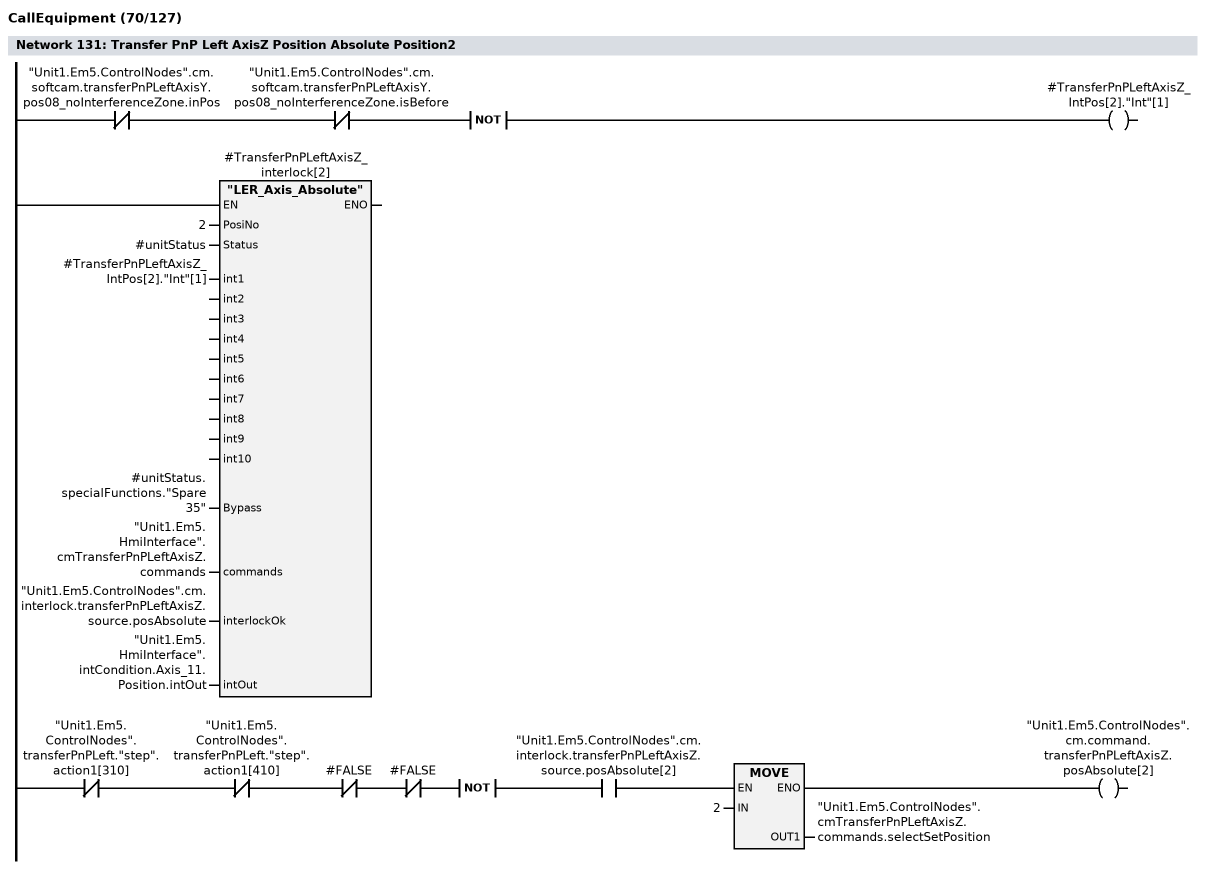
   RUNG wire#powerrail
      I_Contact( "Unit1.Em5.ControlNodes".cm.softcam.transferPnPLeftAxisY.pos08_noInterferenceZone.inPos )
      I_Contact( "Unit1.Em5.ControlNodes".cm.softcam.transferPnPLeftAxisY.pos08_noInterferenceZone.isBefore )
      Not()
      Coil( #TransferPnPLeftAxisZ_IntPos[2]."Int"[1] )
   END_RUNG
   RUNG wire#powerrail
      #TransferPnPLeftAxisZ_interlock[2](PosiNo := 2, Status := #unitStatus, int1 := #TransferPnPLeftAxisZ_IntPos[2]."Int"[1], int2 :=, int3 :=, int4 :=, int5 :=, int6 :=, int7 :=, int8 :=, int9 :=, int10 :=, Bypass := #unitStatus.specialFunctions."Spare 35", commands := "Unit1.Em5.HmiInterface".cmTransferPnPLeftAxisZ.commands, interlockOk := "Unit1.Em5.ControlNodes".cm.interlock.transferPnPLeftAxisZ.source.posAbsolute, intOut := "Unit1.Em5.HmiInterface".intCondition.Axis_11.Position.intOut)
   END_RUNG
   RUNG wire#powerrail
      I_Contact( "Unit1.Em5.ControlNodes".transferPnPLeft."step".action1[310] )
      I_Contact( "Unit1.Em5.ControlNodes".transferPnPLeft."step".action1[410] )
      I_Contact( #FALSE )
      I_Contact( #FALSE )
      Not()
      Contact( "Unit1.Em5.ControlNodes".cm.interlock.transferPnPLeftAxisZ.source.posAbsolute[2] )
      Move(in := 2, out1 => "Unit1.Em5.ControlNodes".cmTransferPnPLeftAxisZ.commands.selectSetPosition)
      Coil( "Unit1.Em5.ControlNodes".cm.command.transferPnPLeftAxisZ.posAbsolute[2] )
   END_RUNG
   // the same network as SCL:
   #TransferPnPLeftAxisZ_IntPos[2]."Int"[1] := NOT (NOT "Unit1.Em5.ControlNodes".cm.softcam.transferPnPLeftAxisY.pos08_noInterferenceZone.inPos AND NOT "Unit1.Em5.ControlNodes".cm.softcam.transferPnPLeftAxisY.pos08_noInterferenceZone.isBefore);
   #TransferPnPLeftAxisZ_interlock[2](PosiNo := 2,   // "LER_Axis_Absolute"
                           Status := #unitStatus,
                           int1 := #TransferPnPLeftAxisZ_IntPos[2]."Int"[1],
                           Bypass := #unitStatus.specialFunctions."Spare 35",
                           commands := "Unit1.Em5.HmiInterface".cmTransferPnPLeftAxisZ.commands,
                           interlockOk := "Unit1.Em5.ControlNodes".cm.interlock.transferPnPLeftAxisZ.source.posAbsolute,
                           intOut := "Unit1.Em5.HmiInterface".intCondition.Axis_11.Position.intOut);
   #_w1 := NOT (NOT "Unit1.Em5.ControlNodes".transferPnPLeft."step".action1[310] AND NOT "Unit1.Em5.ControlNodes".transferPnPLeft."step".action1[410] AND NOT #FALSE AND NOT #FALSE) AND "Unit1.Em5.ControlNodes".cm.interlock.transferPnPLeftAxisZ.source.posAbsolute[2];
   IF #_w1 THEN "Unit1.Em5.ControlNodes".cmTransferPnPLeftAxisZ.commands.selectSetPosition := 2; END_IF;
   "Unit1.Em5.ControlNodes".cm.command.transferPnPLeftAxisZ.posAbsolute[2] := #_w1;
END_REGION

REGION Network 132: Transfer PnP Left AxisZ Position Absolute Position3
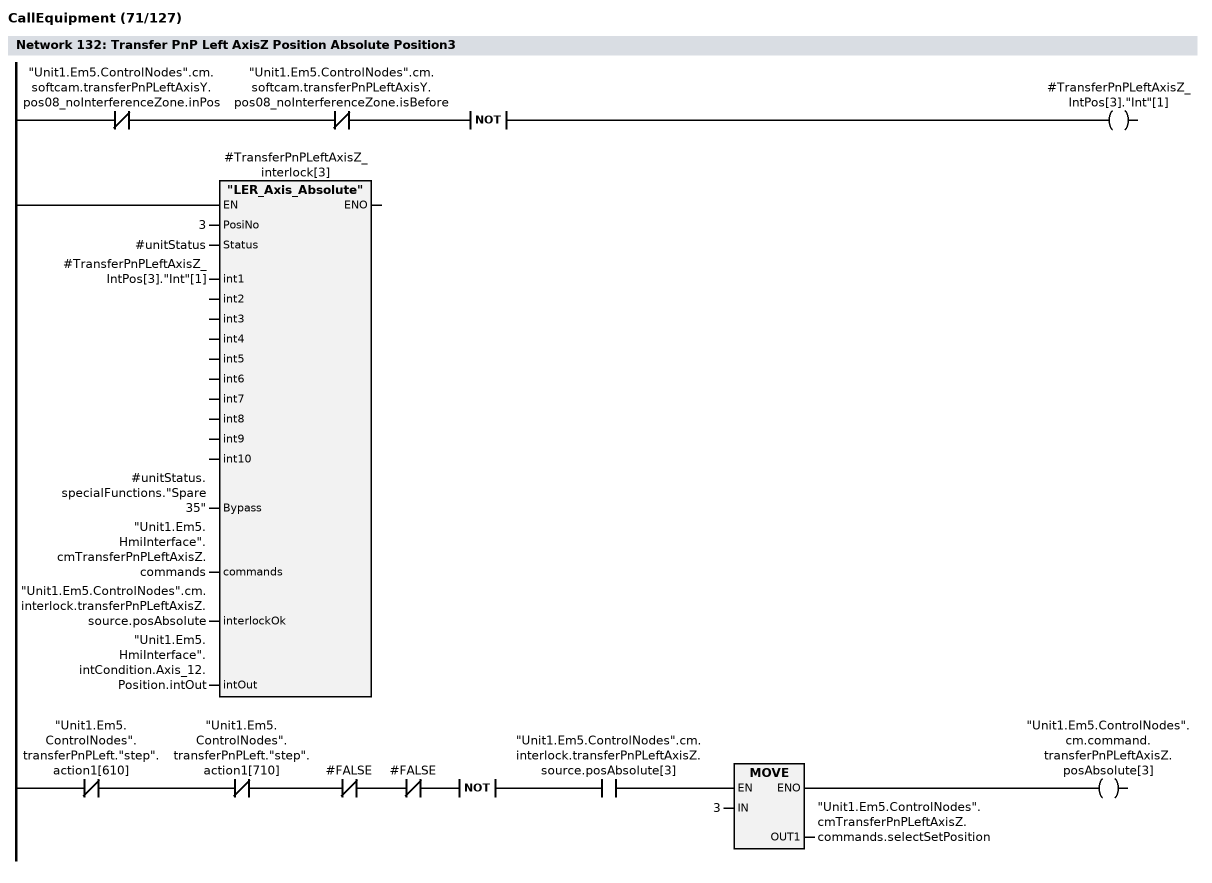
   RUNG wire#powerrail
      I_Contact( "Unit1.Em5.ControlNodes".cm.softcam.transferPnPLeftAxisY.pos08_noInterferenceZone.inPos )
      I_Contact( "Unit1.Em5.ControlNodes".cm.softcam.transferPnPLeftAxisY.pos08_noInterferenceZone.isBefore )
      Not()
      Coil( #TransferPnPLeftAxisZ_IntPos[3]."Int"[1] )
   END_RUNG
   RUNG wire#powerrail
      #TransferPnPLeftAxisZ_interlock[3](PosiNo := 3, Status := #unitStatus, int1 := #TransferPnPLeftAxisZ_IntPos[3]."Int"[1], int2 :=, int3 :=, int4 :=, int5 :=, int6 :=, int7 :=, int8 :=, int9 :=, int10 :=, Bypass := #unitStatus.specialFunctions."Spare 35", commands := "Unit1.Em5.HmiInterface".cmTransferPnPLeftAxisZ.commands, interlockOk := "Unit1.Em5.ControlNodes".cm.interlock.transferPnPLeftAxisZ.source.posAbsolute, intOut := "Unit1.Em5.HmiInterface".intCondition.Axis_12.Position.intOut)
   END_RUNG
   RUNG wire#powerrail
      I_Contact( "Unit1.Em5.ControlNodes".transferPnPLeft."step".action1[610] )
      I_Contact( "Unit1.Em5.ControlNodes".transferPnPLeft."step".action1[710] )
      I_Contact( #FALSE )
      I_Contact( #FALSE )
      Not()
      Contact( "Unit1.Em5.ControlNodes".cm.interlock.transferPnPLeftAxisZ.source.posAbsolute[3] )
      Move(in := 3, out1 => "Unit1.Em5.ControlNodes".cmTransferPnPLeftAxisZ.commands.selectSetPosition)
      Coil( "Unit1.Em5.ControlNodes".cm.command.transferPnPLeftAxisZ.posAbsolute[3] )
   END_RUNG
   // the same network as SCL:
   #TransferPnPLeftAxisZ_IntPos[3]."Int"[1] := NOT (NOT "Unit1.Em5.ControlNodes".cm.softcam.transferPnPLeftAxisY.pos08_noInterferenceZone.inPos AND NOT "Unit1.Em5.ControlNodes".cm.softcam.transferPnPLeftAxisY.pos08_noInterferenceZone.isBefore);
   #TransferPnPLeftAxisZ_interlock[3](PosiNo := 3,   // "LER_Axis_Absolute"
                           Status := #unitStatus,
                           int1 := #TransferPnPLeftAxisZ_IntPos[3]."Int"[1],
                           Bypass := #unitStatus.specialFunctions."Spare 35",
                           commands := "Unit1.Em5.HmiInterface".cmTransferPnPLeftAxisZ.commands,
                           interlockOk := "Unit1.Em5.ControlNodes".cm.interlock.transferPnPLeftAxisZ.source.posAbsolute,
                           intOut := "Unit1.Em5.HmiInterface".intCondition.Axis_12.Position.intOut);
   #_w1 := NOT (NOT "Unit1.Em5.ControlNodes".transferPnPLeft."step".action1[610] AND NOT "Unit1.Em5.ControlNodes".transferPnPLeft."step".action1[710] AND NOT #FALSE AND NOT #FALSE) AND "Unit1.Em5.ControlNodes".cm.interlock.transferPnPLeftAxisZ.source.posAbsolute[3];
   IF #_w1 THEN "Unit1.Em5.ControlNodes".cmTransferPnPLeftAxisZ.commands.selectSetPosition := 3; END_IF;
   "Unit1.Em5.ControlNodes".cm.command.transferPnPLeftAxisZ.posAbsolute[3] := #_w1;
END_REGION

REGION Network 133: Transfer PnP Left AxisZ Position Absolute Position4
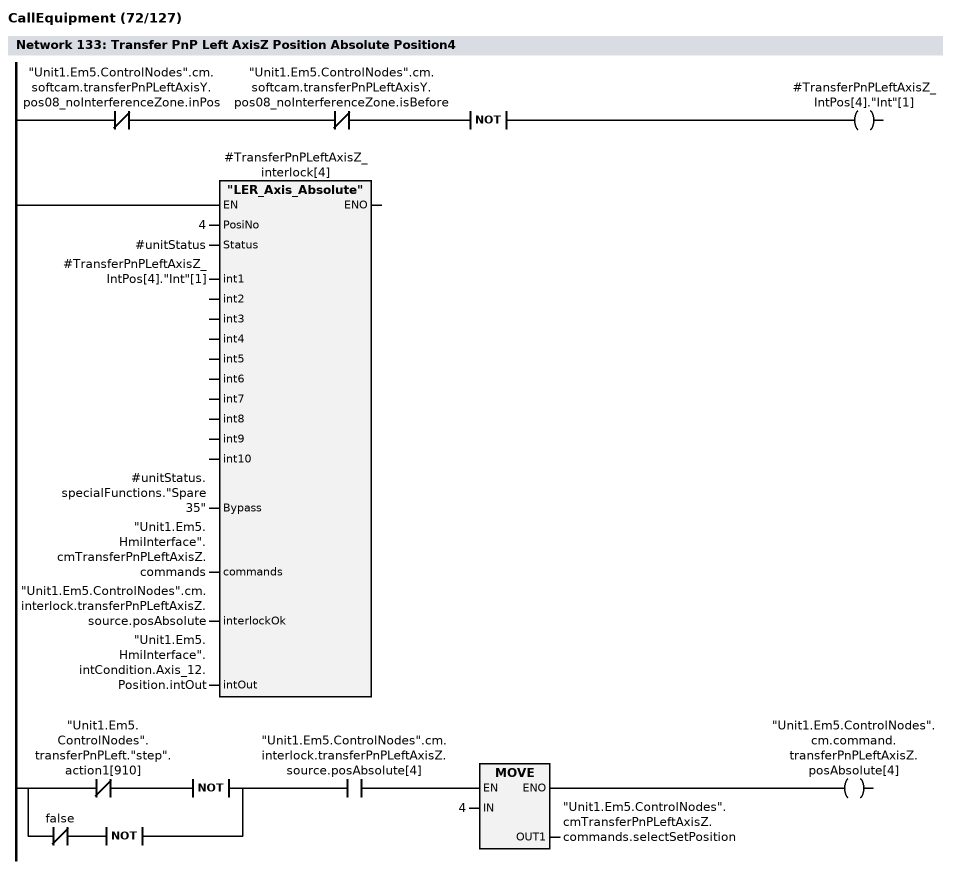
   RUNG wire#powerrail
      I_Contact( "Unit1.Em5.ControlNodes".cm.softcam.transferPnPLeftAxisY.pos08_noInterferenceZone.inPos )
      I_Contact( "Unit1.Em5.ControlNodes".cm.softcam.transferPnPLeftAxisY.pos08_noInterferenceZone.isBefore )
      Not()
      Coil( #TransferPnPLeftAxisZ_IntPos[4]."Int"[1] )
   END_RUNG
   RUNG wire#powerrail
      #TransferPnPLeftAxisZ_interlock[4](PosiNo := 4, Status := #unitStatus, int1 := #TransferPnPLeftAxisZ_IntPos[4]."Int"[1], int2 :=, int3 :=, int4 :=, int5 :=, int6 :=, int7 :=, int8 :=, int9 :=, int10 :=, Bypass := #unitStatus.specialFunctions."Spare 35", commands := "Unit1.Em5.HmiInterface".cmTransferPnPLeftAxisZ.commands, interlockOk := "Unit1.Em5.ControlNodes".cm.interlock.transferPnPLeftAxisZ.source.posAbsolute, intOut := "Unit1.Em5.HmiInterface".intCondition.Axis_12.Position.intOut)
   END_RUNG
   RUNG wire#powerrail
      I_Contact( "Unit1.Em5.ControlNodes".transferPnPLeft."step".action1[910] )
      Not()
      wire#w1
      Contact( "Unit1.Em5.ControlNodes".cm.interlock.transferPnPLeftAxisZ.source.posAbsolute[4] )
      Move(in := 4, out1 => "Unit1.Em5.ControlNodes".cmTransferPnPLeftAxisZ.commands.selectSetPosition)
      Coil( "Unit1.Em5.ControlNodes".cm.command.transferPnPLeftAxisZ.posAbsolute[4] )
   END_RUNG
   RUNG wire#powerrail
      I_Contact( false )
      Not()
   END_RUNG wire#w1
   // the same network as SCL:
   #TransferPnPLeftAxisZ_IntPos[4]."Int"[1] := NOT (NOT "Unit1.Em5.ControlNodes".cm.softcam.transferPnPLeftAxisY.pos08_noInterferenceZone.inPos AND NOT "Unit1.Em5.ControlNodes".cm.softcam.transferPnPLeftAxisY.pos08_noInterferenceZone.isBefore);
   #TransferPnPLeftAxisZ_interlock[4](PosiNo := 4,   // "LER_Axis_Absolute"
                           Status := #unitStatus,
                           int1 := #TransferPnPLeftAxisZ_IntPos[4]."Int"[1],
                           Bypass := #unitStatus.specialFunctions."Spare 35",
                           commands := "Unit1.Em5.HmiInterface".cmTransferPnPLeftAxisZ.commands,
                           interlockOk := "Unit1.Em5.ControlNodes".cm.interlock.transferPnPLeftAxisZ.source.posAbsolute,
                           intOut := "Unit1.Em5.HmiInterface".intCondition.Axis_12.Position.intOut);
   #_w1 := (NOT (NOT "Unit1.Em5.ControlNodes".transferPnPLeft."step".action1[910]) OR NOT (NOT false)) AND "Unit1.Em5.ControlNodes".cm.interlock.transferPnPLeftAxisZ.source.posAbsolute[4];
   IF #_w1 THEN "Unit1.Em5.ControlNodes".cmTransferPnPLeftAxisZ.commands.selectSetPosition := 4; END_IF;
   "Unit1.Em5.ControlNodes".cm.command.transferPnPLeftAxisZ.posAbsolute[4] := #_w1;
END_REGION

REGION Network 134: Transfer PnP Left AxisZ Position Absolute Position5
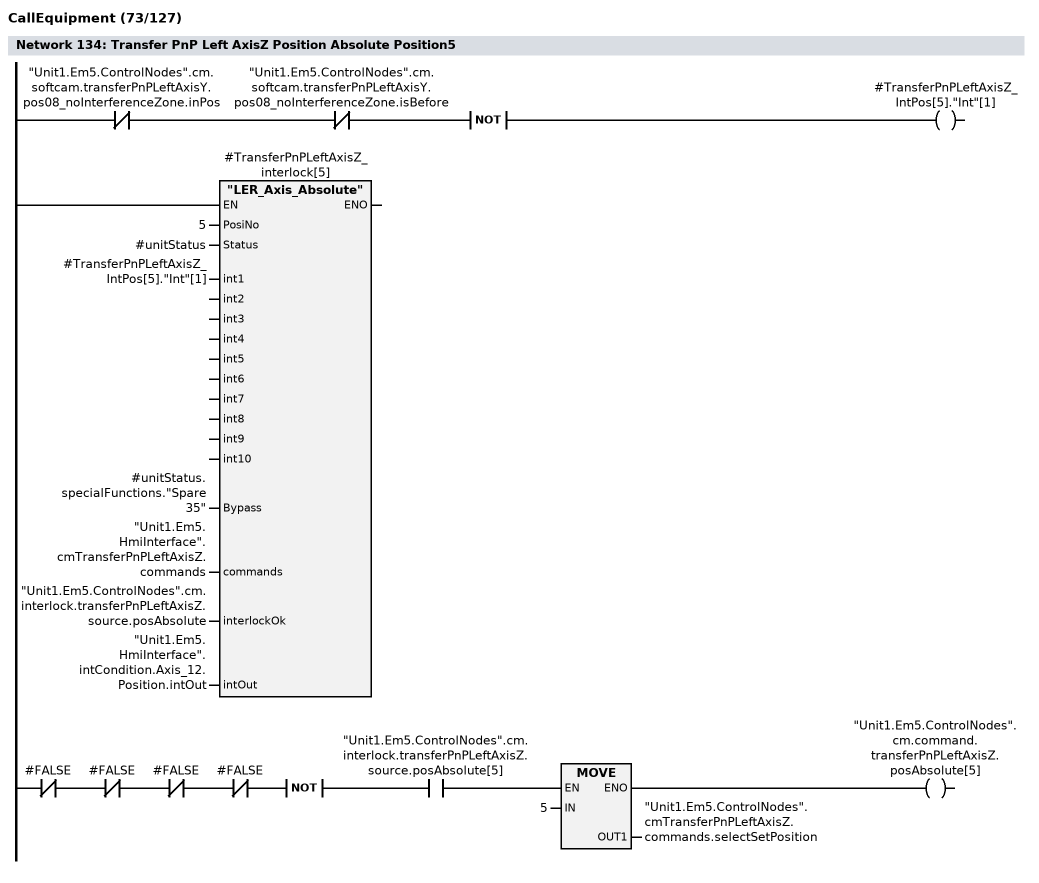
   RUNG wire#powerrail
      I_Contact( "Unit1.Em5.ControlNodes".cm.softcam.transferPnPLeftAxisY.pos08_noInterferenceZone.inPos )
      I_Contact( "Unit1.Em5.ControlNodes".cm.softcam.transferPnPLeftAxisY.pos08_noInterferenceZone.isBefore )
      Not()
      Coil( #TransferPnPLeftAxisZ_IntPos[5]."Int"[1] )
   END_RUNG
   RUNG wire#powerrail
      #TransferPnPLeftAxisZ_interlock[5](PosiNo := 5, Status := #unitStatus, int1 := #TransferPnPLeftAxisZ_IntPos[5]."Int"[1], int2 :=, int3 :=, int4 :=, int5 :=, int6 :=, int7 :=, int8 :=, int9 :=, int10 :=, Bypass := #unitStatus.specialFunctions."Spare 35", commands := "Unit1.Em5.HmiInterface".cmTransferPnPLeftAxisZ.commands, interlockOk := "Unit1.Em5.ControlNodes".cm.interlock.transferPnPLeftAxisZ.source.posAbsolute, intOut := "Unit1.Em5.HmiInterface".intCondition.Axis_12.Position.intOut)
   END_RUNG
   RUNG wire#powerrail
      I_Contact( #FALSE )
      I_Contact( #FALSE )
      I_Contact( #FALSE )
      I_Contact( #FALSE )
      Not()
      Contact( "Unit1.Em5.ControlNodes".cm.interlock.transferPnPLeftAxisZ.source.posAbsolute[5] )
      Move(in := 5, out1 => "Unit1.Em5.ControlNodes".cmTransferPnPLeftAxisZ.commands.selectSetPosition)
      Coil( "Unit1.Em5.ControlNodes".cm.command.transferPnPLeftAxisZ.posAbsolute[5] )
   END_RUNG
   // the same network as SCL:
   #TransferPnPLeftAxisZ_IntPos[5]."Int"[1] := NOT (NOT "Unit1.Em5.ControlNodes".cm.softcam.transferPnPLeftAxisY.pos08_noInterferenceZone.inPos AND NOT "Unit1.Em5.ControlNodes".cm.softcam.transferPnPLeftAxisY.pos08_noInterferenceZone.isBefore);
   #TransferPnPLeftAxisZ_interlock[5](PosiNo := 5,   // "LER_Axis_Absolute"
                           Status := #unitStatus,
                           int1 := #TransferPnPLeftAxisZ_IntPos[5]."Int"[1],
                           Bypass := #unitStatus.specialFunctions."Spare 35",
                           commands := "Unit1.Em5.HmiInterface".cmTransferPnPLeftAxisZ.commands,
                           interlockOk := "Unit1.Em5.ControlNodes".cm.interlock.transferPnPLeftAxisZ.source.posAbsolute,
                           intOut := "Unit1.Em5.HmiInterface".intCondition.Axis_12.Position.intOut);
   #_w1 := NOT (NOT #FALSE AND NOT #FALSE AND NOT #FALSE AND NOT #FALSE) AND "Unit1.Em5.ControlNodes".cm.interlock.transferPnPLeftAxisZ.source.posAbsolute[5];
   IF #_w1 THEN "Unit1.Em5.ControlNodes".cmTransferPnPLeftAxisZ.commands.selectSetPosition := 5; END_IF;
   "Unit1.Em5.ControlNodes".cm.command.transferPnPLeftAxisZ.posAbsolute[5] := #_w1;
END_REGION

REGION Network 135: Transfer PnP Left AxisZ Position Absolute Position7
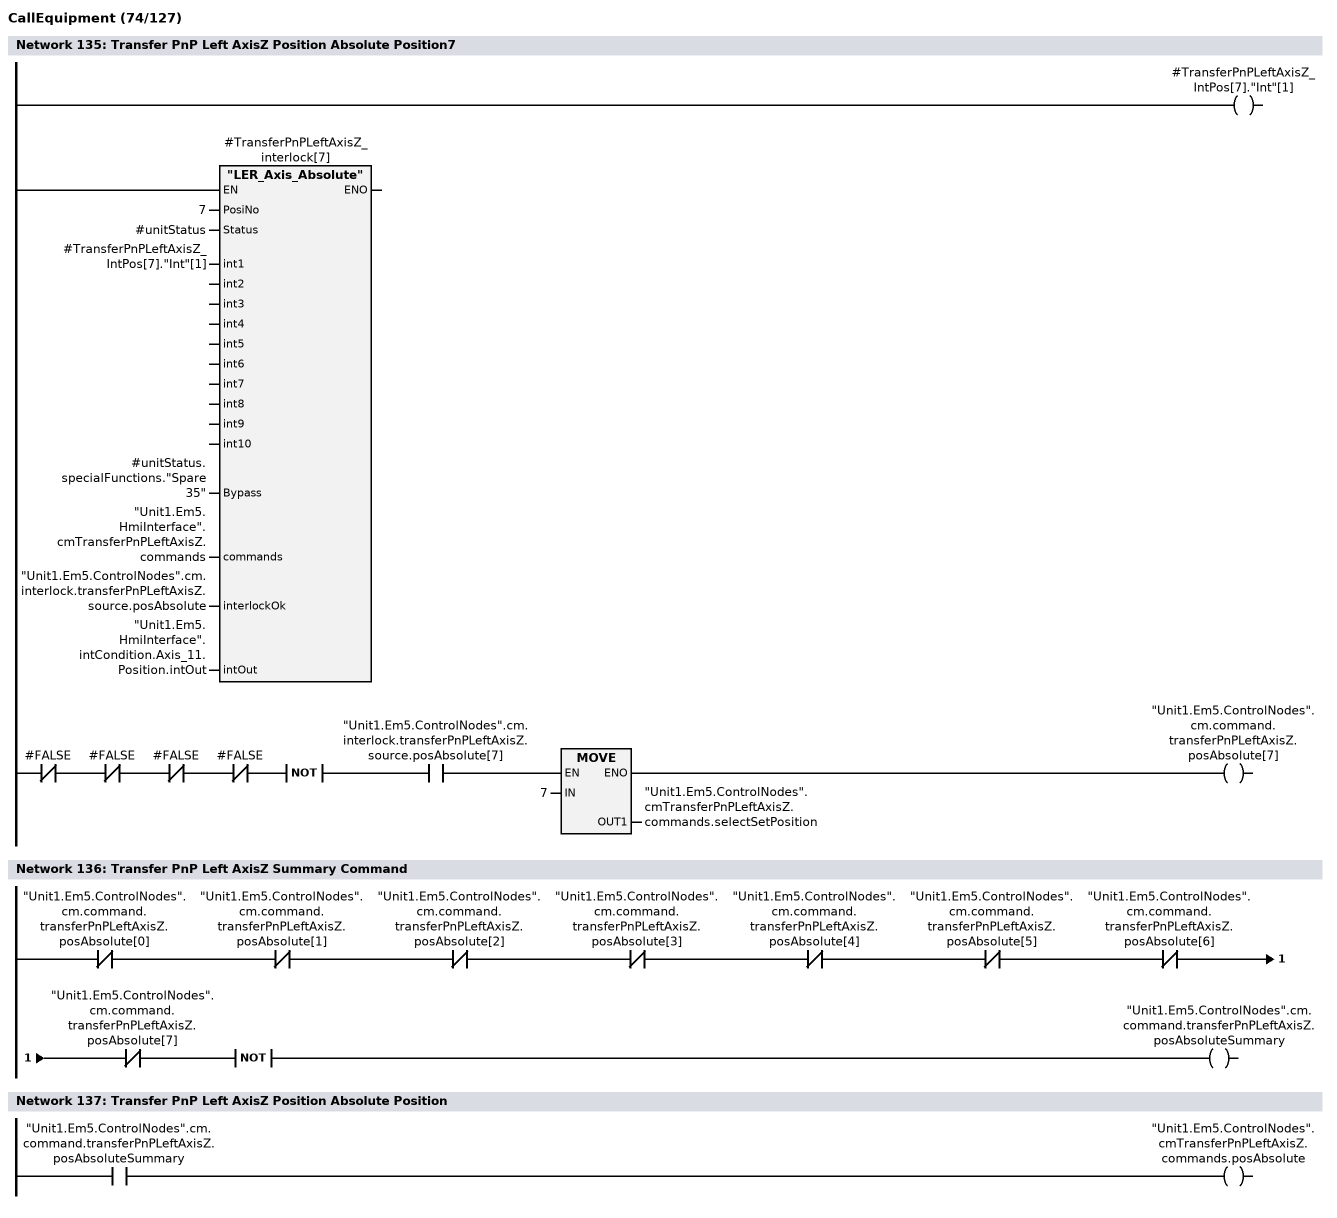
   RUNG wire#powerrail
      Coil( #TransferPnPLeftAxisZ_IntPos[7]."Int"[1] )
   END_RUNG
   RUNG wire#powerrail
      #TransferPnPLeftAxisZ_interlock[7](PosiNo := 7, Status := #unitStatus, int1 := #TransferPnPLeftAxisZ_IntPos[7]."Int"[1], int2 :=, int3 :=, int4 :=, int5 :=, int6 :=, int7 :=, int8 :=, int9 :=, int10 :=, Bypass := #unitStatus.specialFunctions."Spare 35", commands := "Unit1.Em5.HmiInterface".cmTransferPnPLeftAxisZ.commands, interlockOk := "Unit1.Em5.ControlNodes".cm.interlock.transferPnPLeftAxisZ.source.posAbsolute, intOut := "Unit1.Em5.HmiInterface".intCondition.Axis_11.Position.intOut)
   END_RUNG
   RUNG wire#powerrail
      I_Contact( #FALSE )
      I_Contact( #FALSE )
      I_Contact( #FALSE )
      I_Contact( #FALSE )
      Not()
      Contact( "Unit1.Em5.ControlNodes".cm.interlock.transferPnPLeftAxisZ.source.posAbsolute[7] )
      Move(in := 7, out1 => "Unit1.Em5.ControlNodes".cmTransferPnPLeftAxisZ.commands.selectSetPosition)
      Coil( "Unit1.Em5.ControlNodes".cm.command.transferPnPLeftAxisZ.posAbsolute[7] )
   END_RUNG
   // the same network as SCL:
   #TransferPnPLeftAxisZ_IntPos[7]."Int"[1] := TRUE;
   #TransferPnPLeftAxisZ_interlock[7](PosiNo := 7,   // "LER_Axis_Absolute"
                           Status := #unitStatus,
                           int1 := #TransferPnPLeftAxisZ_IntPos[7]."Int"[1],
                           Bypass := #unitStatus.specialFunctions."Spare 35",
                           commands := "Unit1.Em5.HmiInterface".cmTransferPnPLeftAxisZ.commands,
                           interlockOk := "Unit1.Em5.ControlNodes".cm.interlock.transferPnPLeftAxisZ.source.posAbsolute,
                           intOut := "Unit1.Em5.HmiInterface".intCondition.Axis_11.Position.intOut);
   #_w1 := NOT (NOT #FALSE AND NOT #FALSE AND NOT #FALSE AND NOT #FALSE) AND "Unit1.Em5.ControlNodes".cm.interlock.transferPnPLeftAxisZ.source.posAbsolute[7];
   IF #_w1 THEN "Unit1.Em5.ControlNodes".cmTransferPnPLeftAxisZ.commands.selectSetPosition := 7; END_IF;
   "Unit1.Em5.ControlNodes".cm.command.transferPnPLeftAxisZ.posAbsolute[7] := #_w1;
END_REGION

REGION Network 136: Transfer PnP Left AxisZ Summary Command
   RUNG wire#powerrail
      I_Contact( "Unit1.Em5.ControlNodes".cm.command.transferPnPLeftAxisZ.posAbsolute[0] )
      I_Contact( "Unit1.Em5.ControlNodes".cm.command.transferPnPLeftAxisZ.posAbsolute[1] )
      I_Contact( "Unit1.Em5.ControlNodes".cm.command.transferPnPLeftAxisZ.posAbsolute[2] )
      I_Contact( "Unit1.Em5.ControlNodes".cm.command.transferPnPLeftAxisZ.posAbsolute[3] )
      I_Contact( "Unit1.Em5.ControlNodes".cm.command.transferPnPLeftAxisZ.posAbsolute[4] )
      I_Contact( "Unit1.Em5.ControlNodes".cm.command.transferPnPLeftAxisZ.posAbsolute[5] )
      I_Contact( "Unit1.Em5.ControlNodes".cm.command.transferPnPLeftAxisZ.posAbsolute[6] )
      I_Contact( "Unit1.Em5.ControlNodes".cm.command.transferPnPLeftAxisZ.posAbsolute[7] )
      Not()
      Coil( "Unit1.Em5.ControlNodes".cm.command.transferPnPLeftAxisZ.posAbsoluteSummary )
   END_RUNG
   // the same network as SCL:
   "Unit1.Em5.ControlNodes".cm.command.transferPnPLeftAxisZ.posAbsoluteSummary := NOT (NOT "Unit1.Em5.ControlNodes".cm.command.transferPnPLeftAxisZ.posAbsolute[0] AND NOT "Unit1.Em5.ControlNodes".cm.command.transferPnPLeftAxisZ.posAbsolute[1] AND NOT "Unit1.Em5.ControlNodes".cm.command.transferPnPLeftAxisZ.posAbsolute[2] AND NOT "Unit1.Em5.ControlNodes".cm.command.transferPnPLeftAxisZ.posAbsolute[3] AND NOT "Unit1.Em5.ControlNodes".cm.command.transferPnPLeftAxisZ.posAbsolute[4] AND NOT "Unit1.Em5.ControlNodes".cm.command.transferPnPLeftAxisZ.posAbsolute[5] AND NOT "Unit1.Em5.ControlNodes".cm.command.transferPnPLeftAxisZ.posAbsolute[6] AND NOT "Unit1.Em5.ControlNodes".cm.command.transferPnPLeftAxisZ.posAbsolute[7]);
END_REGION

REGION Network 137: Transfer PnP Left AxisZ Position Absolute Position
   RUNG wire#powerrail
      Contact( "Unit1.Em5.ControlNodes".cm.command.transferPnPLeftAxisZ.posAbsoluteSummary )
      Coil( "Unit1.Em5.ControlNodes".cmTransferPnPLeftAxisZ.commands.posAbsolute )
   END_RUNG
   // the same network as SCL:
   "Unit1.Em5.ControlNodes".cmTransferPnPLeftAxisZ.commands.posAbsolute := "Unit1.Em5.ControlNodes".cm.command.transferPnPLeftAxisZ.posAbsoluteSummary;
END_REGION

REGION Network 138: Transfer PnP Left AxisZ Interlock Summary
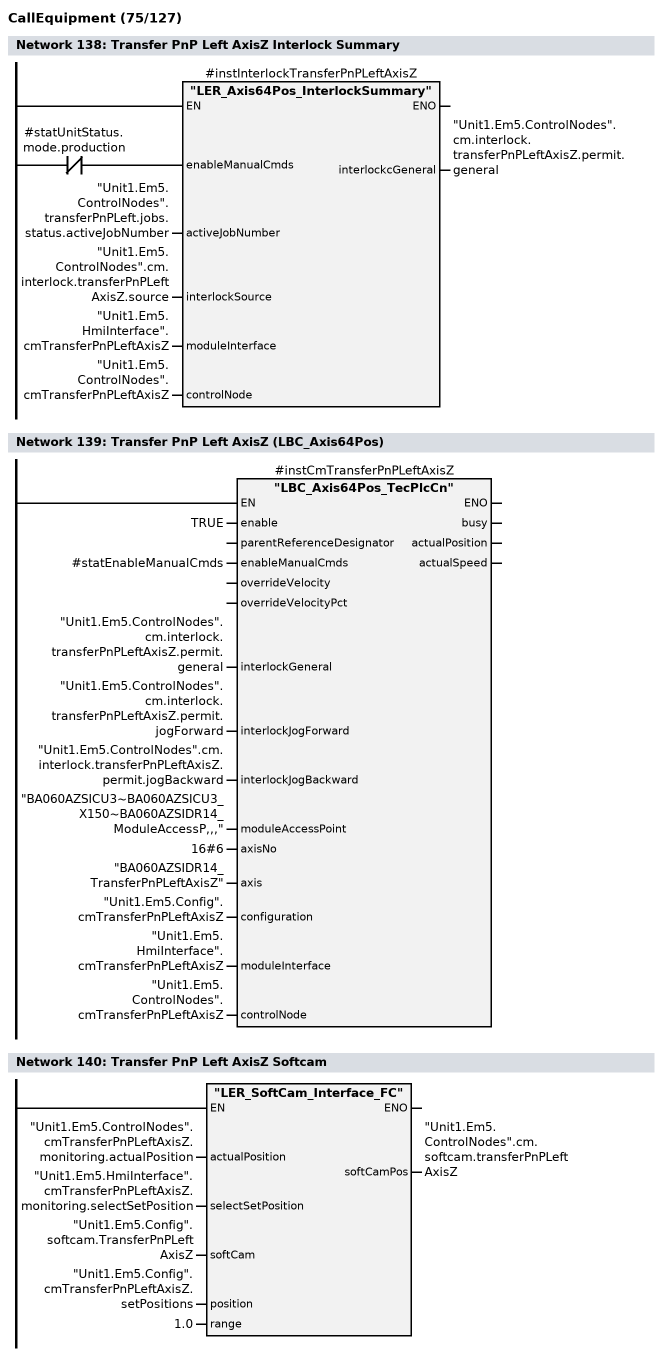
   RUNG wire#powerrail
      #instInterlockTransferPnPLeftAxisZ(enableManualCmds := wire#w1, activeJobNumber := "Unit1.Em5.ControlNodes".transferPnPLeft.jobs.status.activeJobNumber, interlockSource := "Unit1.Em5.ControlNodes".cm.interlock.transferPnPLeftAxisZ.source, moduleInterface := "Unit1.Em5.HmiInterface".cmTransferPnPLeftAxisZ, controlNode := "Unit1.Em5.ControlNodes".cmTransferPnPLeftAxisZ, interlockcGeneral => "Unit1.Em5.ControlNodes".cm.interlock.transferPnPLeftAxisZ.permit.general)
   END_RUNG
   RUNG wire#powerrail
      I_Contact( #statUnitStatus.mode.production )
   END_RUNG wire#w1
   // the same network as SCL:
   #instInterlockTransferPnPLeftAxisZ(enableManualCmds := NOT #statUnitStatus.mode.production,   // "LER_Axis64Pos_InterlockSummary"
                           activeJobNumber := "Unit1.Em5.ControlNodes".transferPnPLeft.jobs.status.activeJobNumber,
                           interlockSource := "Unit1.Em5.ControlNodes".cm.interlock.transferPnPLeftAxisZ.source,
                           moduleInterface := "Unit1.Em5.HmiInterface".cmTransferPnPLeftAxisZ,
                           controlNode := "Unit1.Em5.ControlNodes".cmTransferPnPLeftAxisZ,
                           interlockcGeneral => "Unit1.Em5.ControlNodes".cm.interlock.transferPnPLeftAxisZ.permit.general);
END_REGION

REGION Network 139: Transfer PnP Left AxisZ (LBC_Axis64Pos)
   RUNG wire#powerrail
      #instCmTransferPnPLeftAxisZ(enable := TRUE, parentReferenceDesignator :=, enableManualCmds := #statEnableManualCmds, overrideVelocity :=, overrideVelocityPct :=, interlockGeneral := "Unit1.Em5.ControlNodes".cm.interlock.transferPnPLeftAxisZ.permit.general, interlockJogForward := "Unit1.Em5.ControlNodes".cm.interlock.transferPnPLeftAxisZ.permit.jogForward, interlockJogBackward := "Unit1.Em5.ControlNodes".cm.interlock.transferPnPLeftAxisZ.permit.jogBackward, moduleAccessPoint := "BA060AZSICU3~BA060AZSICU3_X150~BA060AZSIDR14_ModuleAccessP,,,", axisNo := 16#6, axis := "BA060AZSIDR14_TransferPnPLeftAxisZ", configuration := "Unit1.Em5.Config".cmTransferPnPLeftAxisZ, moduleInterface := "Unit1.Em5.HmiInterface".cmTransferPnPLeftAxisZ, controlNode := "Unit1.Em5.ControlNodes".cmTransferPnPLeftAxisZ, busy =>, actualPosition =>, actualSpeed =>)
   END_RUNG
   // the same network as SCL:
   #instCmTransferPnPLeftAxisZ(enable := TRUE,   // "LBC_Axis64Pos_TecPlcCn"
                           enableManualCmds := #statEnableManualCmds,
                           interlockGeneral := "Unit1.Em5.ControlNodes".cm.interlock.transferPnPLeftAxisZ.permit.general,
                           interlockJogForward := "Unit1.Em5.ControlNodes".cm.interlock.transferPnPLeftAxisZ.permit.jogForward,
                           interlockJogBackward := "Unit1.Em5.ControlNodes".cm.interlock.transferPnPLeftAxisZ.permit.jogBackward,
                           moduleAccessPoint := "BA060AZSICU3~BA060AZSICU3_X150~BA060AZSIDR14_ModuleAccessP,,,",
                           axisNo := 16#6,
                           axis := "BA060AZSIDR14_TransferPnPLeftAxisZ",
                           configuration := "Unit1.Em5.Config".cmTransferPnPLeftAxisZ,
                           moduleInterface := "Unit1.Em5.HmiInterface".cmTransferPnPLeftAxisZ,
                           controlNode := "Unit1.Em5.ControlNodes".cmTransferPnPLeftAxisZ);
END_REGION

REGION Network 140: Transfer PnP Left AxisZ Softcam
   RUNG wire#powerrail
      "LER_SoftCam_Interface_FC"(actualPosition := "Unit1.Em5.ControlNodes".cmTransferPnPLeftAxisZ.monitoring.actualPosition, selectSetPosition := "Unit1.Em5.HmiInterface".cmTransferPnPLeftAxisZ.monitoring.selectSetPosition, softCam := "Unit1.Em5.Config".softcam.TransferPnPLeftAxisZ, position := "Unit1.Em5.Config".cmTransferPnPLeftAxisZ.setPositions, range := 1.0, softCamPos => "Unit1.Em5.ControlNodes".cm.softcam.transferPnPLeftAxisZ)
   END_RUNG
   // the same network as SCL:
   "LER_SoftCam_Interface_FC"(actualPosition := "Unit1.Em5.ControlNodes".cmTransferPnPLeftAxisZ.monitoring.actualPosition,
                           selectSetPosition := "Unit1.Em5.HmiInterface".cmTransferPnPLeftAxisZ.monitoring.selectSetPosition,
                           softCam := "Unit1.Em5.Config".softcam.TransferPnPLeftAxisZ,
                           position := "Unit1.Em5.Config".cmTransferPnPLeftAxisZ.setPositions,
                           range := 1.0,
                           softCamPos => "Unit1.Em5.ControlNodes".cm.softcam.transferPnPLeftAxisZ);
END_REGION

REGION Network 142: Transfer P&P Right X-Axis Upload Actual Current And Torque Values
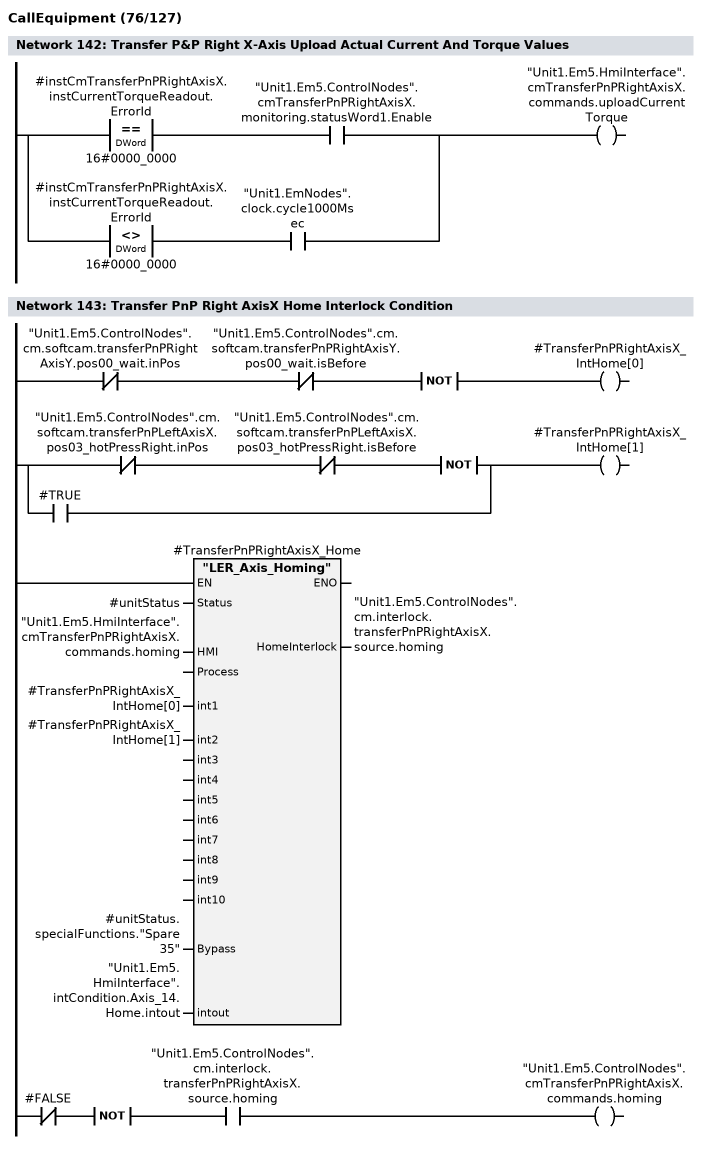
   RUNG wire#powerrail
      { S7_Templates := "SrcType := DWord" } EQ_Contact(in1 := #instCmTransferPnPRightAxisX.instCurrentTorqueReadout.ErrorId, in2 := 16#0000_0000)
      Contact( "Unit1.Em5.ControlNodes".cmTransferPnPRightAxisX.monitoring.statusWord1.Enable )
      wire#w1
      Coil( "Unit1.Em5.HmiInterface".cmTransferPnPRightAxisX.commands.uploadCurrentTorque )
   END_RUNG
   RUNG wire#powerrail
      { S7_Templates := "SrcType := DWord" } NE_Contact(in1 := #instCmTransferPnPRightAxisX.instCurrentTorqueReadout.ErrorId, in2 := 16#0000_0000)
      Contact( "Unit1.EmNodes".clock.cycle1000Msec )
   END_RUNG wire#w1
   // the same network as SCL:
   "Unit1.Em5.HmiInterface".cmTransferPnPRightAxisX.commands.uploadCurrentTorque := ((#instCmTransferPnPRightAxisX.instCurrentTorqueReadout.ErrorId = 16#0000_0000) AND "Unit1.Em5.ControlNodes".cmTransferPnPRightAxisX.monitoring.statusWord1.Enable) OR ((#instCmTransferPnPRightAxisX.instCurrentTorqueReadout.ErrorId <> 16#0000_0000) AND "Unit1.EmNodes".clock.cycle1000Msec);
END_REGION

REGION Network 143: Transfer PnP Right AxisX Home Interlock Condition
   RUNG wire#powerrail
      I_Contact( "Unit1.Em5.ControlNodes".cm.softcam.transferPnPRightAxisY.pos00_wait.inPos )
      I_Contact( "Unit1.Em5.ControlNodes".cm.softcam.transferPnPRightAxisY.pos00_wait.isBefore )
      Not()
      Coil( #TransferPnPRightAxisX_IntHome[0] )
   END_RUNG
   RUNG wire#powerrail
      I_Contact( "Unit1.Em5.ControlNodes".cm.softcam.transferPnPLeftAxisX.pos03_hotPressRight.inPos )
      I_Contact( "Unit1.Em5.ControlNodes".cm.softcam.transferPnPLeftAxisX.pos03_hotPressRight.isBefore )
      Not()
      wire#w1
      Coil( #TransferPnPRightAxisX_IntHome[1] )
   END_RUNG
   RUNG wire#powerrail
      Contact( #TRUE )
   END_RUNG wire#w1
   RUNG wire#powerrail
      #TransferPnPRightAxisX_Home(Status := #unitStatus, HMI := "Unit1.Em5.HmiInterface".cmTransferPnPRightAxisX.commands.homing, Process :=, int1 := #TransferPnPRightAxisX_IntHome[0], int2 := #TransferPnPRightAxisX_IntHome[1], int3 :=, int4 :=, int5 :=, int6 :=, int7 :=, int8 :=, int9 :=, int10 :=, Bypass := #unitStatus.specialFunctions."Spare 35", intout := "Unit1.Em5.HmiInterface".intCondition.Axis_14.Home.intout, HomeInterlock => "Unit1.Em5.ControlNodes".cm.interlock.transferPnPRightAxisX.source.homing)
   END_RUNG
   RUNG wire#powerrail
      I_Contact( #FALSE )
      Not()
      Contact( "Unit1.Em5.ControlNodes".cm.interlock.transferPnPRightAxisX.source.homing )
      Coil( "Unit1.Em5.ControlNodes".cmTransferPnPRightAxisX.commands.homing )
   END_RUNG
   // the same network as SCL:
   #TransferPnPRightAxisX_IntHome[0] := NOT (NOT "Unit1.Em5.ControlNodes".cm.softcam.transferPnPRightAxisY.pos00_wait.inPos AND NOT "Unit1.Em5.ControlNodes".cm.softcam.transferPnPRightAxisY.pos00_wait.isBefore);
   #TransferPnPRightAxisX_IntHome[1] := NOT (NOT "Unit1.Em5.ControlNodes".cm.softcam.transferPnPLeftAxisX.pos03_hotPressRight.inPos AND NOT "Unit1.Em5.ControlNodes".cm.softcam.transferPnPLeftAxisX.pos03_hotPressRight.isBefore) OR #TRUE;
   #TransferPnPRightAxisX_Home(Status := #unitStatus,   // "LER_Axis_Homing"
                           HMI := "Unit1.Em5.HmiInterface".cmTransferPnPRightAxisX.commands.homing,
                           int1 := #TransferPnPRightAxisX_IntHome[0],
                           int2 := #TransferPnPRightAxisX_IntHome[1],
                           Bypass := #unitStatus.specialFunctions."Spare 35",
                           intout := "Unit1.Em5.HmiInterface".intCondition.Axis_14.Home.intout,
                           HomeInterlock => "Unit1.Em5.ControlNodes".cm.interlock.transferPnPRightAxisX.source.homing);
   "Unit1.Em5.ControlNodes".cmTransferPnPRightAxisX.commands.homing := NOT (NOT #FALSE) AND "Unit1.Em5.ControlNodes".cm.interlock.transferPnPRightAxisX.source.homing;
END_REGION

REGION Network 144: Transfer PnP Right AxisX JOG Interlock Condition
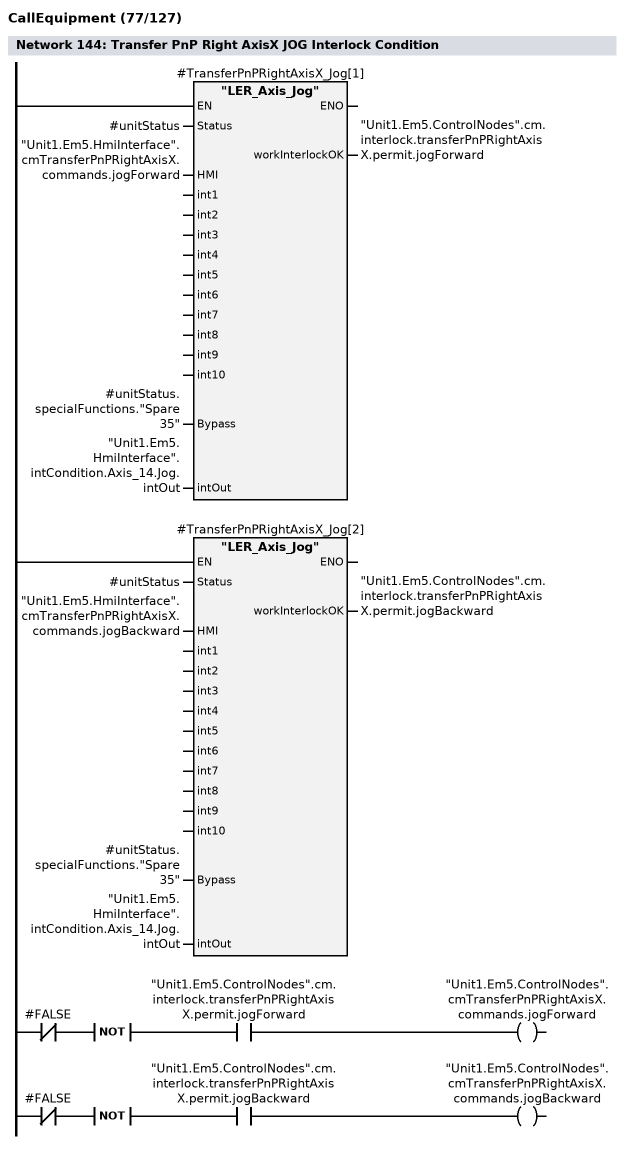
   RUNG wire#powerrail
      #TransferPnPRightAxisX_Jog[1](Status := #unitStatus, HMI := "Unit1.Em5.HmiInterface".cmTransferPnPRightAxisX.commands.jogForward, int1 :=, int2 :=, int3 :=, int4 :=, int5 :=, int6 :=, int7 :=, int8 :=, int9 :=, int10 :=, Bypass := #unitStatus.specialFunctions."Spare 35", intOut := "Unit1.Em5.HmiInterface".intCondition.Axis_14.Jog.intOut, workInterlockOK => "Unit1.Em5.ControlNodes".cm.interlock.transferPnPRightAxisX.permit.jogForward)
   END_RUNG
   RUNG wire#powerrail
      #TransferPnPRightAxisX_Jog[2](Status := #unitStatus, HMI := "Unit1.Em5.HmiInterface".cmTransferPnPRightAxisX.commands.jogBackward, int1 :=, int2 :=, int3 :=, int4 :=, int5 :=, int6 :=, int7 :=, int8 :=, int9 :=, int10 :=, Bypass := #unitStatus.specialFunctions."Spare 35", intOut := "Unit1.Em5.HmiInterface".intCondition.Axis_14.Jog.intOut, workInterlockOK => "Unit1.Em5.ControlNodes".cm.interlock.transferPnPRightAxisX.permit.jogBackward)
   END_RUNG
   RUNG wire#powerrail
      I_Contact( #FALSE )
      Not()
      Contact( "Unit1.Em5.ControlNodes".cm.interlock.transferPnPRightAxisX.permit.jogForward )
      Coil( "Unit1.Em5.ControlNodes".cmTransferPnPRightAxisX.commands.jogForward )
   END_RUNG
   RUNG wire#powerrail
      I_Contact( #FALSE )
      Not()
      Contact( "Unit1.Em5.ControlNodes".cm.interlock.transferPnPRightAxisX.permit.jogBackward )
      Coil( "Unit1.Em5.ControlNodes".cmTransferPnPRightAxisX.commands.jogBackward )
   END_RUNG
   // the same network as SCL:
   #TransferPnPRightAxisX_Jog[1](Status := #unitStatus,   // "LER_Axis_Jog"
                           HMI := "Unit1.Em5.HmiInterface".cmTransferPnPRightAxisX.commands.jogForward,
                           Bypass := #unitStatus.specialFunctions."Spare 35",
                           intOut := "Unit1.Em5.HmiInterface".intCondition.Axis_14.Jog.intOut,
                           workInterlockOK => "Unit1.Em5.ControlNodes".cm.interlock.transferPnPRightAxisX.permit.jogForward);
   #TransferPnPRightAxisX_Jog[2](Status := #unitStatus,   // "LER_Axis_Jog"
                           HMI := "Unit1.Em5.HmiInterface".cmTransferPnPRightAxisX.commands.jogBackward,
                           Bypass := #unitStatus.specialFunctions."Spare 35",
                           intOut := "Unit1.Em5.HmiInterface".intCondition.Axis_14.Jog.intOut,
                           workInterlockOK => "Unit1.Em5.ControlNodes".cm.interlock.transferPnPRightAxisX.permit.jogBackward);
   "Unit1.Em5.ControlNodes".cmTransferPnPRightAxisX.commands.jogForward := NOT (NOT #FALSE) AND "Unit1.Em5.ControlNodes".cm.interlock.transferPnPRightAxisX.permit.jogForward;
   "Unit1.Em5.ControlNodes".cmTransferPnPRightAxisX.commands.jogBackward := NOT (NOT #FALSE) AND "Unit1.Em5.ControlNodes".cm.interlock.transferPnPRightAxisX.permit.jogBackward;
END_REGION

REGION Network 145: Transfer PnP Right AxisX Position Absolute Position0 [wait-laser]
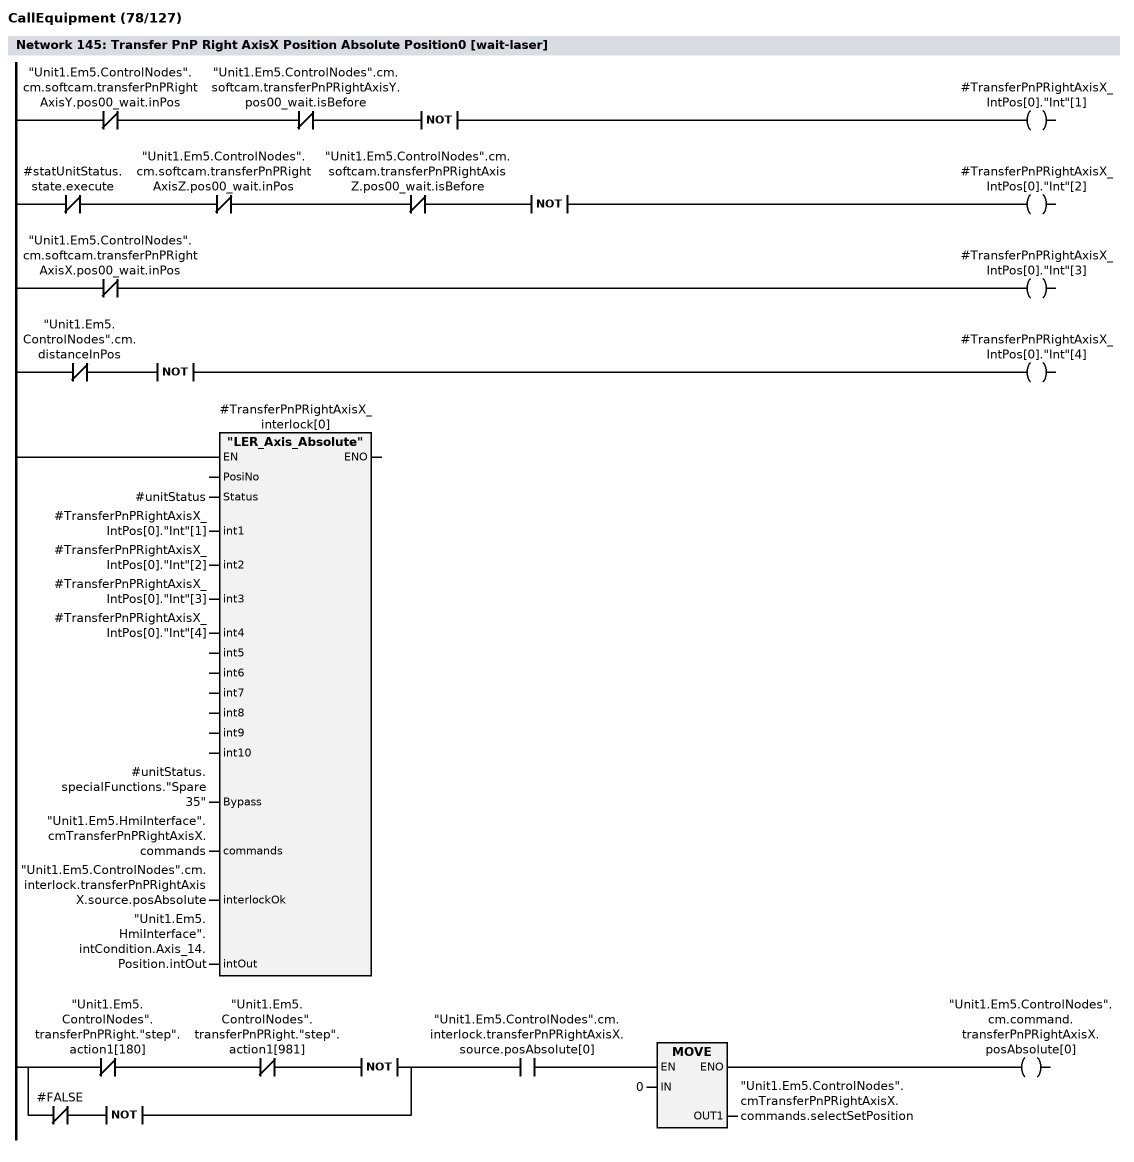
   RUNG wire#powerrail
      I_Contact( "Unit1.Em5.ControlNodes".cm.softcam.transferPnPRightAxisY.pos00_wait.inPos )
      I_Contact( "Unit1.Em5.ControlNodes".cm.softcam.transferPnPRightAxisY.pos00_wait.isBefore )
      Not()
      Coil( #TransferPnPRightAxisX_IntPos[0]."Int"[1] )
   END_RUNG
   RUNG wire#powerrail
      I_Contact( #statUnitStatus.state.execute )
      I_Contact( "Unit1.Em5.ControlNodes".cm.softcam.transferPnPRightAxisZ.pos00_wait.inPos )
      I_Contact( "Unit1.Em5.ControlNodes".cm.softcam.transferPnPRightAxisZ.pos00_wait.isBefore )
      Not()
      Coil( #TransferPnPRightAxisX_IntPos[0]."Int"[2] )
   END_RUNG
   RUNG wire#powerrail
      I_Contact( "Unit1.Em5.ControlNodes".cm.softcam.transferPnPRightAxisX.pos00_wait.inPos )
      Coil( #TransferPnPRightAxisX_IntPos[0]."Int"[3] )
   END_RUNG
   RUNG wire#powerrail
      I_Contact( "Unit1.Em5.ControlNodes".cm.distanceInPos )
      Not()
      Coil( #TransferPnPRightAxisX_IntPos[0]."Int"[4] )
   END_RUNG
   RUNG wire#powerrail
      #TransferPnPRightAxisX_interlock[0](PosiNo :=, Status := #unitStatus, int1 := #TransferPnPRightAxisX_IntPos[0]."Int"[1], int2 := #TransferPnPRightAxisX_IntPos[0]."Int"[2], int3 := #TransferPnPRightAxisX_IntPos[0]."Int"[3], int4 := #TransferPnPRightAxisX_IntPos[0]."Int"[4], int5 :=, int6 :=, int7 :=, int8 :=, int9 :=, int10 :=, Bypass := #unitStatus.specialFunctions."Spare 35", commands := "Unit1.Em5.HmiInterface".cmTransferPnPRightAxisX.commands, interlockOk := "Unit1.Em5.ControlNodes".cm.interlock.transferPnPRightAxisX.source.posAbsolute, intOut := "Unit1.Em5.HmiInterface".intCondition.Axis_14.Position.intOut)
   END_RUNG
   RUNG wire#powerrail
      I_Contact( "Unit1.Em5.ControlNodes".transferPnPRight."step".action1[180] )
      I_Contact( "Unit1.Em5.ControlNodes".transferPnPRight."step".action1[981] )
      Not()
      wire#w1
      Contact( "Unit1.Em5.ControlNodes".cm.interlock.transferPnPRightAxisX.source.posAbsolute[0] )
      Move(in := 0, out1 => "Unit1.Em5.ControlNodes".cmTransferPnPRightAxisX.commands.selectSetPosition)
      Coil( "Unit1.Em5.ControlNodes".cm.command.transferPnPRightAxisX.posAbsolute[0] )
   END_RUNG
   RUNG wire#powerrail
      I_Contact( #FALSE )
      Not()
   END_RUNG wire#w1
   // the same network as SCL:
   #TransferPnPRightAxisX_IntPos[0]."Int"[1] := NOT (NOT "Unit1.Em5.ControlNodes".cm.softcam.transferPnPRightAxisY.pos00_wait.inPos AND NOT "Unit1.Em5.ControlNodes".cm.softcam.transferPnPRightAxisY.pos00_wait.isBefore);
   #TransferPnPRightAxisX_IntPos[0]."Int"[2] := NOT (NOT #statUnitStatus.state.execute AND NOT "Unit1.Em5.ControlNodes".cm.softcam.transferPnPRightAxisZ.pos00_wait.inPos AND NOT "Unit1.Em5.ControlNodes".cm.softcam.transferPnPRightAxisZ.pos00_wait.isBefore);
   #TransferPnPRightAxisX_IntPos[0]."Int"[3] := NOT "Unit1.Em5.ControlNodes".cm.softcam.transferPnPRightAxisX.pos00_wait.inPos;
   #TransferPnPRightAxisX_IntPos[0]."Int"[4] := NOT (NOT "Unit1.Em5.ControlNodes".cm.distanceInPos);
   #TransferPnPRightAxisX_interlock[0](Status := #unitStatus,   // "LER_Axis_Absolute"
                           int1 := #TransferPnPRightAxisX_IntPos[0]."Int"[1],
                           int2 := #TransferPnPRightAxisX_IntPos[0]."Int"[2],
                           int3 := #TransferPnPRightAxisX_IntPos[0]."Int"[3],
                           int4 := #TransferPnPRightAxisX_IntPos[0]."Int"[4],
                           Bypass := #unitStatus.specialFunctions."Spare 35",
                           commands := "Unit1.Em5.HmiInterface".cmTransferPnPRightAxisX.commands,
                           interlockOk := "Unit1.Em5.ControlNodes".cm.interlock.transferPnPRightAxisX.source.posAbsolute,
                           intOut := "Unit1.Em5.HmiInterface".intCondition.Axis_14.Position.intOut);
   #_w1 := (NOT (NOT "Unit1.Em5.ControlNodes".transferPnPRight."step".action1[180] AND NOT "Unit1.Em5.ControlNodes".transferPnPRight."step".action1[981]) OR NOT (NOT #FALSE)) AND "Unit1.Em5.ControlNodes".cm.interlock.transferPnPRightAxisX.source.posAbsolute[0];
   IF #_w1 THEN "Unit1.Em5.ControlNodes".cmTransferPnPRightAxisX.commands.selectSetPosition := 0; END_IF;
   "Unit1.Em5.ControlNodes".cm.command.transferPnPRightAxisX.posAbsolute[0] := #_w1;
END_REGION

REGION Network 146: Transfer PnP Right AxisX Position Absolute Position1 [Hipot]
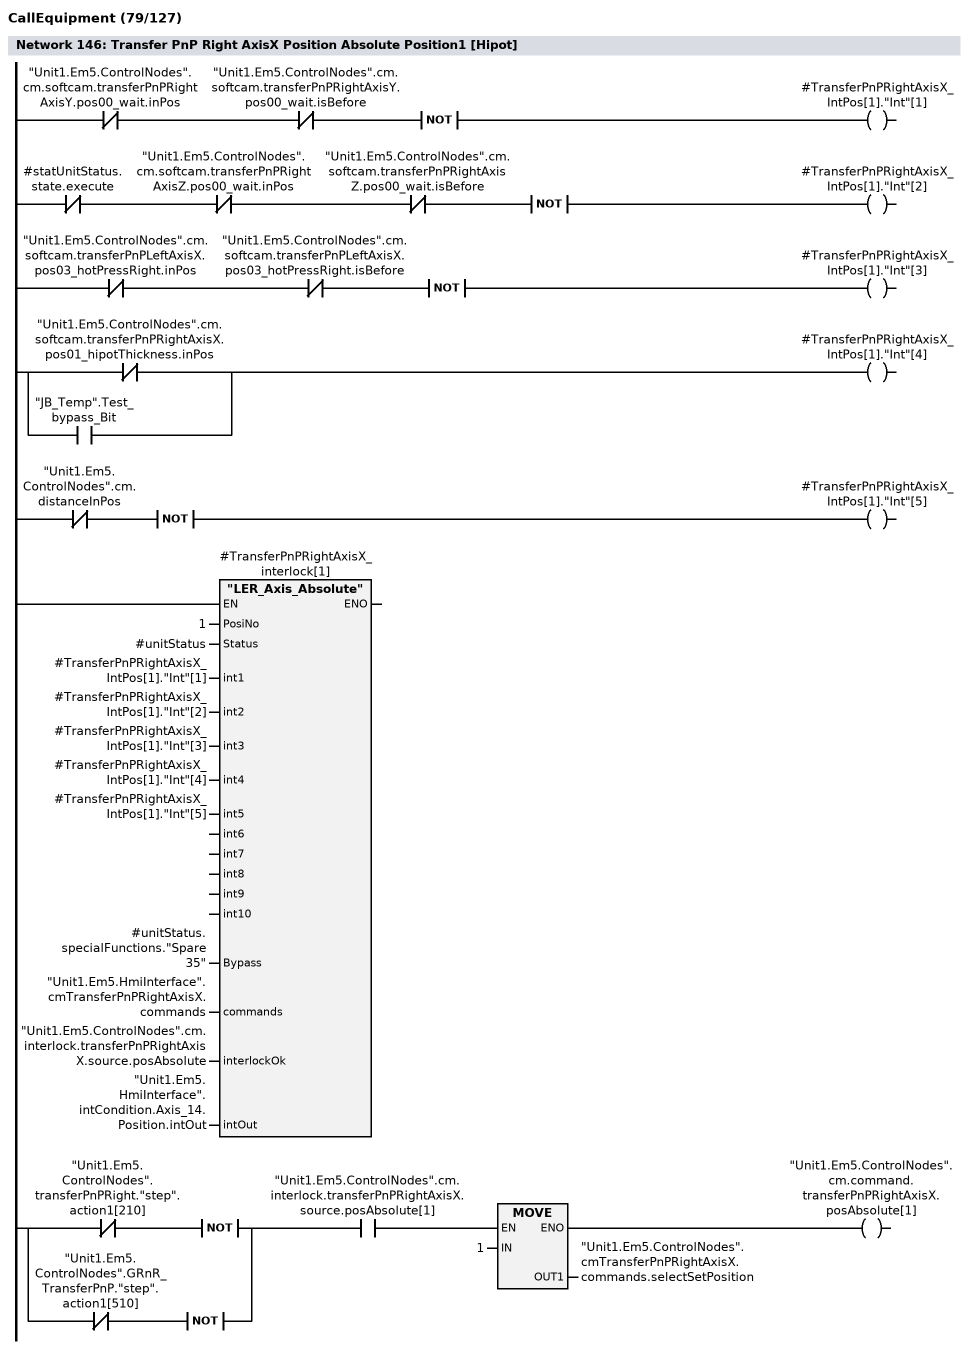
   RUNG wire#powerrail
      I_Contact( "Unit1.Em5.ControlNodes".cm.softcam.transferPnPRightAxisY.pos00_wait.inPos )
      I_Contact( "Unit1.Em5.ControlNodes".cm.softcam.transferPnPRightAxisY.pos00_wait.isBefore )
      Not()
      Coil( #TransferPnPRightAxisX_IntPos[1]."Int"[1] )
   END_RUNG
   RUNG wire#powerrail
      I_Contact( #statUnitStatus.state.execute )
      I_Contact( "Unit1.Em5.ControlNodes".cm.softcam.transferPnPRightAxisZ.pos00_wait.inPos )
      I_Contact( "Unit1.Em5.ControlNodes".cm.softcam.transferPnPRightAxisZ.pos00_wait.isBefore )
      Not()
      Coil( #TransferPnPRightAxisX_IntPos[1]."Int"[2] )
   END_RUNG
   RUNG wire#powerrail
      I_Contact( "Unit1.Em5.ControlNodes".cm.softcam.transferPnPLeftAxisX.pos03_hotPressRight.inPos )
      I_Contact( "Unit1.Em5.ControlNodes".cm.softcam.transferPnPLeftAxisX.pos03_hotPressRight.isBefore )
      Not()
      Coil( #TransferPnPRightAxisX_IntPos[1]."Int"[3] )
   END_RUNG
   RUNG wire#powerrail
      I_Contact( "Unit1.Em5.ControlNodes".cm.softcam.transferPnPRightAxisX.pos01_hipotThickness.inPos )
      wire#w1
      Coil( #TransferPnPRightAxisX_IntPos[1]."Int"[4] )
   END_RUNG
   RUNG wire#powerrail
      Contact( "JB_Temp".Test_bypass_Bit )
   END_RUNG wire#w1
   RUNG wire#powerrail
      I_Contact( "Unit1.Em5.ControlNodes".cm.distanceInPos )
      Not()
      Coil( #TransferPnPRightAxisX_IntPos[1]."Int"[5] )
   END_RUNG
   RUNG wire#powerrail
      #TransferPnPRightAxisX_interlock[1](PosiNo := 1, Status := #unitStatus, int1 := #TransferPnPRightAxisX_IntPos[1]."Int"[1], int2 := #TransferPnPRightAxisX_IntPos[1]."Int"[2], int3 := #TransferPnPRightAxisX_IntPos[1]."Int"[3], int4 := #TransferPnPRightAxisX_IntPos[1]."Int"[4], int5 := #TransferPnPRightAxisX_IntPos[1]."Int"[5], int6 :=, int7 :=, int8 :=, int9 :=, int10 :=, Bypass := #unitStatus.specialFunctions."Spare 35", commands := "Unit1.Em5.HmiInterface".cmTransferPnPRightAxisX.commands, interlockOk := "Unit1.Em5.ControlNodes".cm.interlock.transferPnPRightAxisX.source.posAbsolute, intOut := "Unit1.Em5.HmiInterface".intCondition.Axis_14.Position.intOut)
   END_RUNG
   RUNG wire#powerrail
      I_Contact( "Unit1.Em5.ControlNodes".transferPnPRight."step".action1[210] )
      Not()
      wire#w2
      Contact( "Unit1.Em5.ControlNodes".cm.interlock.transferPnPRightAxisX.source.posAbsolute[1] )
      Move(in := 1, out1 => "Unit1.Em5.ControlNodes".cmTransferPnPRightAxisX.commands.selectSetPosition)
      Coil( "Unit1.Em5.ControlNodes".cm.command.transferPnPRightAxisX.posAbsolute[1] )
   END_RUNG
   RUNG wire#powerrail
      I_Contact( "Unit1.Em5.ControlNodes".GRnR_TransferPnP."step".action1[510] )
      Not()
   END_RUNG wire#w2
   // the same network as SCL:
   #TransferPnPRightAxisX_IntPos[1]."Int"[1] := NOT (NOT "Unit1.Em5.ControlNodes".cm.softcam.transferPnPRightAxisY.pos00_wait.inPos AND NOT "Unit1.Em5.ControlNodes".cm.softcam.transferPnPRightAxisY.pos00_wait.isBefore);
   #TransferPnPRightAxisX_IntPos[1]."Int"[2] := NOT (NOT #statUnitStatus.state.execute AND NOT "Unit1.Em5.ControlNodes".cm.softcam.transferPnPRightAxisZ.pos00_wait.inPos AND NOT "Unit1.Em5.ControlNodes".cm.softcam.transferPnPRightAxisZ.pos00_wait.isBefore);
   #TransferPnPRightAxisX_IntPos[1]."Int"[3] := NOT (NOT "Unit1.Em5.ControlNodes".cm.softcam.transferPnPLeftAxisX.pos03_hotPressRight.inPos AND NOT "Unit1.Em5.ControlNodes".cm.softcam.transferPnPLeftAxisX.pos03_hotPressRight.isBefore);
   #TransferPnPRightAxisX_IntPos[1]."Int"[4] := NOT "Unit1.Em5.ControlNodes".cm.softcam.transferPnPRightAxisX.pos01_hipotThickness.inPos OR "JB_Temp".Test_bypass_Bit;
   #TransferPnPRightAxisX_IntPos[1]."Int"[5] := NOT (NOT "Unit1.Em5.ControlNodes".cm.distanceInPos);
   #TransferPnPRightAxisX_interlock[1](PosiNo := 1,   // "LER_Axis_Absolute"
                           Status := #unitStatus,
                           int1 := #TransferPnPRightAxisX_IntPos[1]."Int"[1],
                           int2 := #TransferPnPRightAxisX_IntPos[1]."Int"[2],
                           int3 := #TransferPnPRightAxisX_IntPos[1]."Int"[3],
                           int4 := #TransferPnPRightAxisX_IntPos[1]."Int"[4],
                           int5 := #TransferPnPRightAxisX_IntPos[1]."Int"[5],
                           Bypass := #unitStatus.specialFunctions."Spare 35",
                           commands := "Unit1.Em5.HmiInterface".cmTransferPnPRightAxisX.commands,
                           interlockOk := "Unit1.Em5.ControlNodes".cm.interlock.transferPnPRightAxisX.source.posAbsolute,
                           intOut := "Unit1.Em5.HmiInterface".intCondition.Axis_14.Position.intOut);
   #_w1 := (NOT (NOT "Unit1.Em5.ControlNodes".transferPnPRight."step".action1[210]) OR NOT (NOT "Unit1.Em5.ControlNodes".GRnR_TransferPnP."step".action1[510])) AND "Unit1.Em5.ControlNodes".cm.interlock.transferPnPRightAxisX.source.posAbsolute[1];
   IF #_w1 THEN "Unit1.Em5.ControlNodes".cmTransferPnPRightAxisX.commands.selectSetPosition := 1; END_IF;
   "Unit1.Em5.ControlNodes".cm.command.transferPnPRightAxisX.posAbsolute[1] := #_w1;
END_REGION

REGION Network 147: Transfer PnP Right AxisX Position Absolute Position2 [vision]
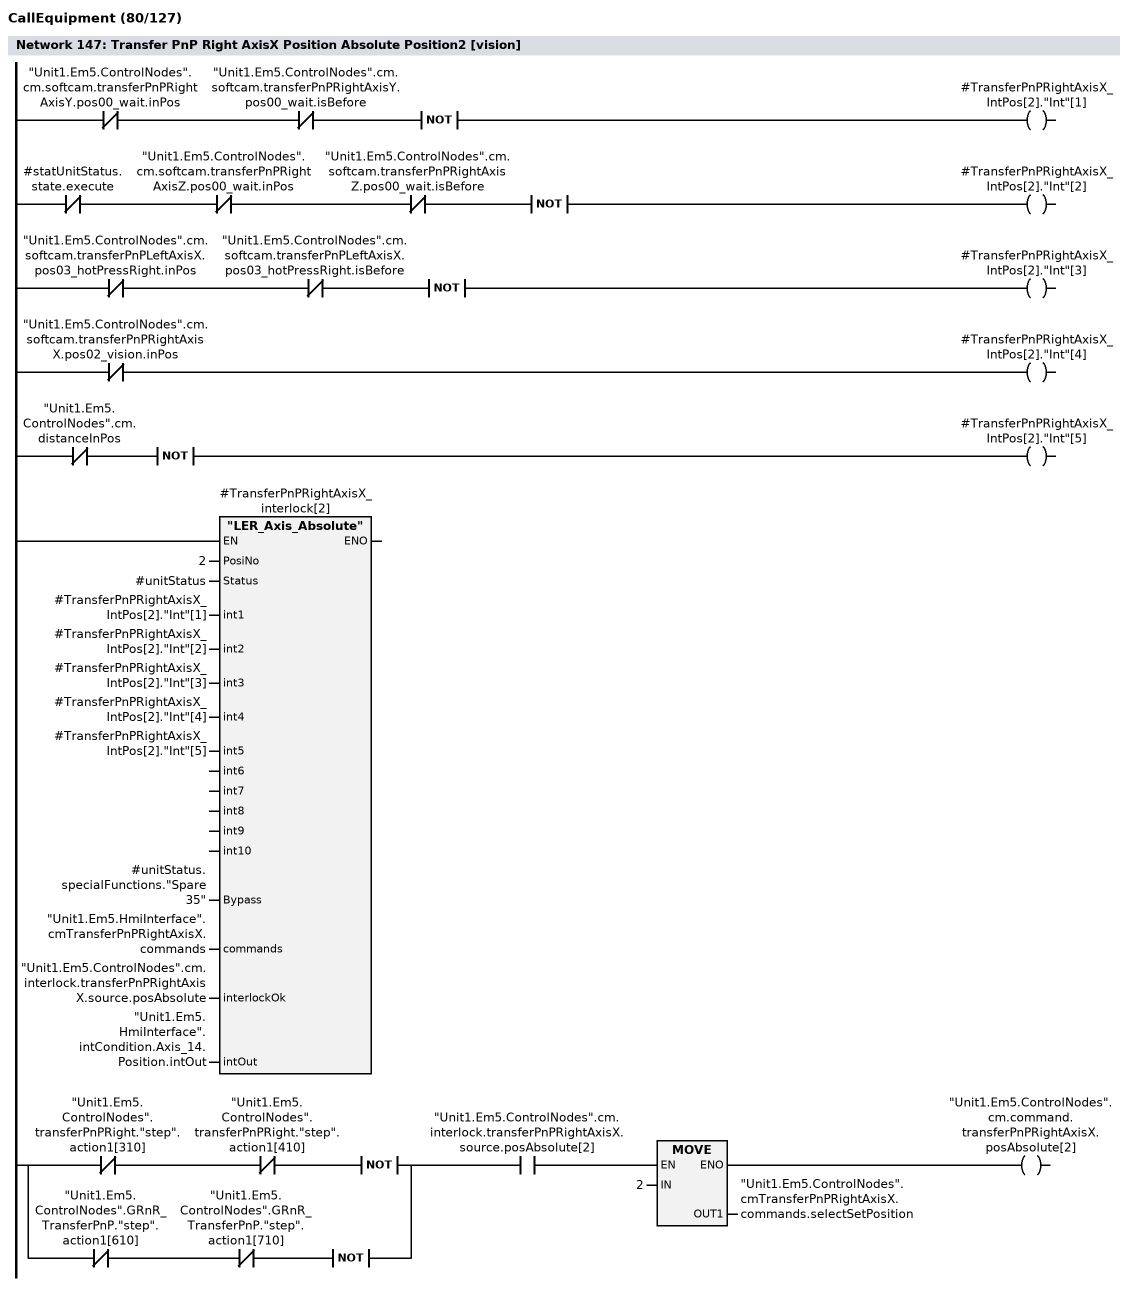
   RUNG wire#powerrail
      I_Contact( "Unit1.Em5.ControlNodes".cm.softcam.transferPnPRightAxisY.pos00_wait.inPos )
      I_Contact( "Unit1.Em5.ControlNodes".cm.softcam.transferPnPRightAxisY.pos00_wait.isBefore )
      Not()
      Coil( #TransferPnPRightAxisX_IntPos[2]."Int"[1] )
   END_RUNG
   RUNG wire#powerrail
      I_Contact( #statUnitStatus.state.execute )
      I_Contact( "Unit1.Em5.ControlNodes".cm.softcam.transferPnPRightAxisZ.pos00_wait.inPos )
      I_Contact( "Unit1.Em5.ControlNodes".cm.softcam.transferPnPRightAxisZ.pos00_wait.isBefore )
      Not()
      Coil( #TransferPnPRightAxisX_IntPos[2]."Int"[2] )
   END_RUNG
   RUNG wire#powerrail
      I_Contact( "Unit1.Em5.ControlNodes".cm.softcam.transferPnPLeftAxisX.pos03_hotPressRight.inPos )
      I_Contact( "Unit1.Em5.ControlNodes".cm.softcam.transferPnPLeftAxisX.pos03_hotPressRight.isBefore )
      Not()
      Coil( #TransferPnPRightAxisX_IntPos[2]."Int"[3] )
   END_RUNG
   RUNG wire#powerrail
      I_Contact( "Unit1.Em5.ControlNodes".cm.softcam.transferPnPRightAxisX.pos02_vision.inPos )
      Coil( #TransferPnPRightAxisX_IntPos[2]."Int"[4] )
   END_RUNG
   RUNG wire#powerrail
      I_Contact( "Unit1.Em5.ControlNodes".cm.distanceInPos )
      Not()
      Coil( #TransferPnPRightAxisX_IntPos[2]."Int"[5] )
   END_RUNG
   RUNG wire#powerrail
      #TransferPnPRightAxisX_interlock[2](PosiNo := 2, Status := #unitStatus, int1 := #TransferPnPRightAxisX_IntPos[2]."Int"[1], int2 := #TransferPnPRightAxisX_IntPos[2]."Int"[2], int3 := #TransferPnPRightAxisX_IntPos[2]."Int"[3], int4 := #TransferPnPRightAxisX_IntPos[2]."Int"[4], int5 := #TransferPnPRightAxisX_IntPos[2]."Int"[5], int6 :=, int7 :=, int8 :=, int9 :=, int10 :=, Bypass := #unitStatus.specialFunctions."Spare 35", commands := "Unit1.Em5.HmiInterface".cmTransferPnPRightAxisX.commands, interlockOk := "Unit1.Em5.ControlNodes".cm.interlock.transferPnPRightAxisX.source.posAbsolute, intOut := "Unit1.Em5.HmiInterface".intCondition.Axis_14.Position.intOut)
   END_RUNG
   RUNG wire#powerrail
      I_Contact( "Unit1.Em5.ControlNodes".transferPnPRight."step".action1[310] )
      I_Contact( "Unit1.Em5.ControlNodes".transferPnPRight."step".action1[410] )
      Not()
      wire#w1
      Contact( "Unit1.Em5.ControlNodes".cm.interlock.transferPnPRightAxisX.source.posAbsolute[2] )
      Move(in := 2, out1 => "Unit1.Em5.ControlNodes".cmTransferPnPRightAxisX.commands.selectSetPosition)
      Coil( "Unit1.Em5.ControlNodes".cm.command.transferPnPRightAxisX.posAbsolute[2] )
   END_RUNG
   RUNG wire#powerrail
      I_Contact( "Unit1.Em5.ControlNodes".GRnR_TransferPnP."step".action1[610] )
      I_Contact( "Unit1.Em5.ControlNodes".GRnR_TransferPnP."step".action1[710] )
      Not()
   END_RUNG wire#w1
   // the same network as SCL:
   #TransferPnPRightAxisX_IntPos[2]."Int"[1] := NOT (NOT "Unit1.Em5.ControlNodes".cm.softcam.transferPnPRightAxisY.pos00_wait.inPos AND NOT "Unit1.Em5.ControlNodes".cm.softcam.transferPnPRightAxisY.pos00_wait.isBefore);
   #TransferPnPRightAxisX_IntPos[2]."Int"[2] := NOT (NOT #statUnitStatus.state.execute AND NOT "Unit1.Em5.ControlNodes".cm.softcam.transferPnPRightAxisZ.pos00_wait.inPos AND NOT "Unit1.Em5.ControlNodes".cm.softcam.transferPnPRightAxisZ.pos00_wait.isBefore);
   #TransferPnPRightAxisX_IntPos[2]."Int"[3] := NOT (NOT "Unit1.Em5.ControlNodes".cm.softcam.transferPnPLeftAxisX.pos03_hotPressRight.inPos AND NOT "Unit1.Em5.ControlNodes".cm.softcam.transferPnPLeftAxisX.pos03_hotPressRight.isBefore);
   #TransferPnPRightAxisX_IntPos[2]."Int"[4] := NOT "Unit1.Em5.ControlNodes".cm.softcam.transferPnPRightAxisX.pos02_vision.inPos;
   #TransferPnPRightAxisX_IntPos[2]."Int"[5] := NOT (NOT "Unit1.Em5.ControlNodes".cm.distanceInPos);
   #TransferPnPRightAxisX_interlock[2](PosiNo := 2,   // "LER_Axis_Absolute"
                           Status := #unitStatus,
                           int1 := #TransferPnPRightAxisX_IntPos[2]."Int"[1],
                           int2 := #TransferPnPRightAxisX_IntPos[2]."Int"[2],
                           int3 := #TransferPnPRightAxisX_IntPos[2]."Int"[3],
                           int4 := #TransferPnPRightAxisX_IntPos[2]."Int"[4],
                           int5 := #TransferPnPRightAxisX_IntPos[2]."Int"[5],
                           Bypass := #unitStatus.specialFunctions."Spare 35",
                           commands := "Unit1.Em5.HmiInterface".cmTransferPnPRightAxisX.commands,
                           interlockOk := "Unit1.Em5.ControlNodes".cm.interlock.transferPnPRightAxisX.source.posAbsolute,
                           intOut := "Unit1.Em5.HmiInterface".intCondition.Axis_14.Position.intOut);
   #_w1 := (NOT (NOT "Unit1.Em5.ControlNodes".transferPnPRight."step".action1[310] AND NOT "Unit1.Em5.ControlNodes".transferPnPRight."step".action1[410]) OR NOT (NOT "Unit1.Em5.ControlNodes".GRnR_TransferPnP."step".action1[610] AND NOT "Unit1.Em5.ControlNodes".GRnR_TransferPnP."step".action1[710])) AND "Unit1.Em5.ControlNodes".cm.interlock.transferPnPRightAxisX.source.posAbsolute[2];
   IF #_w1 THEN "Unit1.Em5.ControlNodes".cmTransferPnPRightAxisX.commands.selectSetPosition := 2; END_IF;
   "Unit1.Em5.ControlNodes".cm.command.transferPnPRightAxisX.posAbsolute[2] := #_w1;
END_REGION

REGION Network 148: Transfer PnP Right AxisX Position Absolute Position3 [laser]
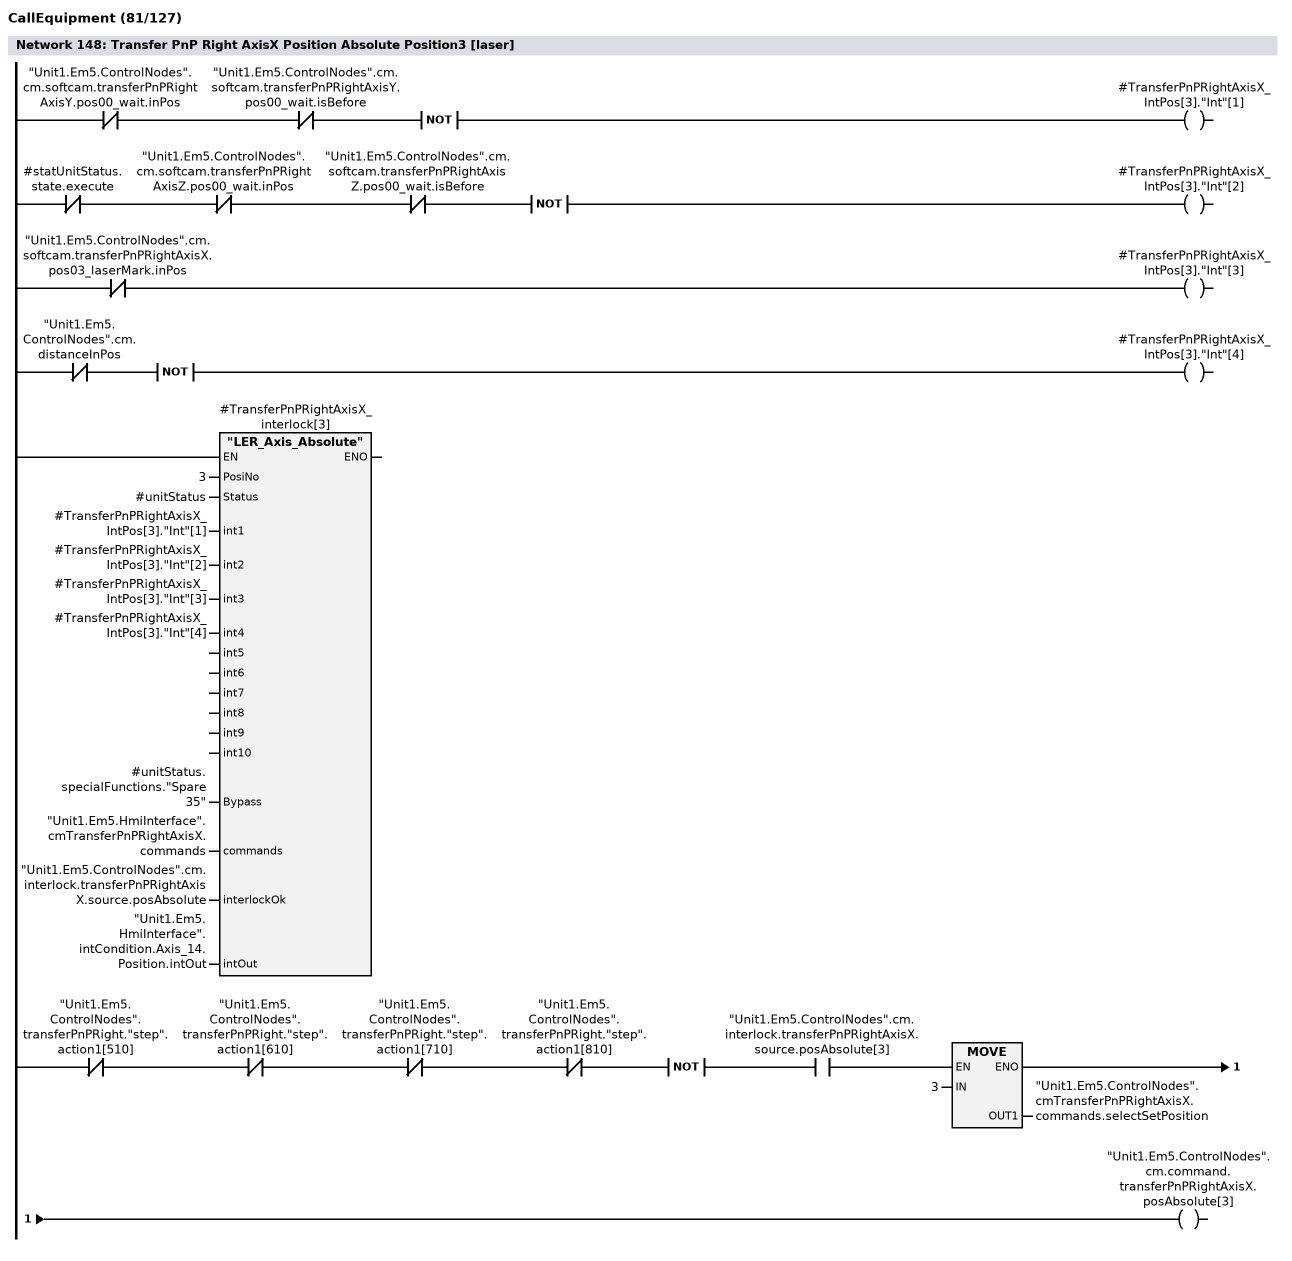
   RUNG wire#powerrail
      I_Contact( "Unit1.Em5.ControlNodes".cm.softcam.transferPnPRightAxisY.pos00_wait.inPos )
      I_Contact( "Unit1.Em5.ControlNodes".cm.softcam.transferPnPRightAxisY.pos00_wait.isBefore )
      Not()
      Coil( #TransferPnPRightAxisX_IntPos[3]."Int"[1] )
   END_RUNG
   RUNG wire#powerrail
      I_Contact( #statUnitStatus.state.execute )
      I_Contact( "Unit1.Em5.ControlNodes".cm.softcam.transferPnPRightAxisZ.pos00_wait.inPos )
      I_Contact( "Unit1.Em5.ControlNodes".cm.softcam.transferPnPRightAxisZ.pos00_wait.isBefore )
      Not()
      Coil( #TransferPnPRightAxisX_IntPos[3]."Int"[2] )
   END_RUNG
   RUNG wire#powerrail
      I_Contact( "Unit1.Em5.ControlNodes".cm.softcam.transferPnPRightAxisX.pos03_laserMark.inPos )
      Coil( #TransferPnPRightAxisX_IntPos[3]."Int"[3] )
   END_RUNG
   RUNG wire#powerrail
      I_Contact( "Unit1.Em5.ControlNodes".cm.distanceInPos )
      Not()
      Coil( #TransferPnPRightAxisX_IntPos[3]."Int"[4] )
   END_RUNG
   RUNG wire#powerrail
      #TransferPnPRightAxisX_interlock[3](PosiNo := 3, Status := #unitStatus, int1 := #TransferPnPRightAxisX_IntPos[3]."Int"[1], int2 := #TransferPnPRightAxisX_IntPos[3]."Int"[2], int3 := #TransferPnPRightAxisX_IntPos[3]."Int"[3], int4 := #TransferPnPRightAxisX_IntPos[3]."Int"[4], int5 :=, int6 :=, int7 :=, int8 :=, int9 :=, int10 :=, Bypass := #unitStatus.specialFunctions."Spare 35", commands := "Unit1.Em5.HmiInterface".cmTransferPnPRightAxisX.commands, interlockOk := "Unit1.Em5.ControlNodes".cm.interlock.transferPnPRightAxisX.source.posAbsolute, intOut := "Unit1.Em5.HmiInterface".intCondition.Axis_14.Position.intOut)
   END_RUNG
   RUNG wire#powerrail
      I_Contact( "Unit1.Em5.ControlNodes".transferPnPRight."step".action1[510] )
      I_Contact( "Unit1.Em5.ControlNodes".transferPnPRight."step".action1[610] )
      I_Contact( "Unit1.Em5.ControlNodes".transferPnPRight."step".action1[710] )
      I_Contact( "Unit1.Em5.ControlNodes".transferPnPRight."step".action1[810] )
      Not()
      Contact( "Unit1.Em5.ControlNodes".cm.interlock.transferPnPRightAxisX.source.posAbsolute[3] )
      Move(in := 3, out1 => "Unit1.Em5.ControlNodes".cmTransferPnPRightAxisX.commands.selectSetPosition)
      Coil( "Unit1.Em5.ControlNodes".cm.command.transferPnPRightAxisX.posAbsolute[3] )
   END_RUNG
   // the same network as SCL:
   #TransferPnPRightAxisX_IntPos[3]."Int"[1] := NOT (NOT "Unit1.Em5.ControlNodes".cm.softcam.transferPnPRightAxisY.pos00_wait.inPos AND NOT "Unit1.Em5.ControlNodes".cm.softcam.transferPnPRightAxisY.pos00_wait.isBefore);
   #TransferPnPRightAxisX_IntPos[3]."Int"[2] := NOT (NOT #statUnitStatus.state.execute AND NOT "Unit1.Em5.ControlNodes".cm.softcam.transferPnPRightAxisZ.pos00_wait.inPos AND NOT "Unit1.Em5.ControlNodes".cm.softcam.transferPnPRightAxisZ.pos00_wait.isBefore);
   #TransferPnPRightAxisX_IntPos[3]."Int"[3] := NOT "Unit1.Em5.ControlNodes".cm.softcam.transferPnPRightAxisX.pos03_laserMark.inPos;
   #TransferPnPRightAxisX_IntPos[3]."Int"[4] := NOT (NOT "Unit1.Em5.ControlNodes".cm.distanceInPos);
   #TransferPnPRightAxisX_interlock[3](PosiNo := 3,   // "LER_Axis_Absolute"
                           Status := #unitStatus,
                           int1 := #TransferPnPRightAxisX_IntPos[3]."Int"[1],
                           int2 := #TransferPnPRightAxisX_IntPos[3]."Int"[2],
                           int3 := #TransferPnPRightAxisX_IntPos[3]."Int"[3],
                           int4 := #TransferPnPRightAxisX_IntPos[3]."Int"[4],
                           Bypass := #unitStatus.specialFunctions."Spare 35",
                           commands := "Unit1.Em5.HmiInterface".cmTransferPnPRightAxisX.commands,
                           interlockOk := "Unit1.Em5.ControlNodes".cm.interlock.transferPnPRightAxisX.source.posAbsolute,
                           intOut := "Unit1.Em5.HmiInterface".intCondition.Axis_14.Position.intOut);
   #_w1 := NOT (NOT "Unit1.Em5.ControlNodes".transferPnPRight."step".action1[510] AND NOT "Unit1.Em5.ControlNodes".transferPnPRight."step".action1[610] AND NOT "Unit1.Em5.ControlNodes".transferPnPRight."step".action1[710] AND NOT "Unit1.Em5.ControlNodes".transferPnPRight."step".action1[810]) AND "Unit1.Em5.ControlNodes".cm.interlock.transferPnPRightAxisX.source.posAbsolute[3];
   IF #_w1 THEN "Unit1.Em5.ControlNodes".cmTransferPnPRightAxisX.commands.selectSetPosition := 3; END_IF;
   "Unit1.Em5.ControlNodes".cm.command.transferPnPRightAxisX.posAbsolute[3] := #_w1;
END_REGION

REGION Network 149: Transfer PnP Right AxisX Position Absolute Position4 [weight]
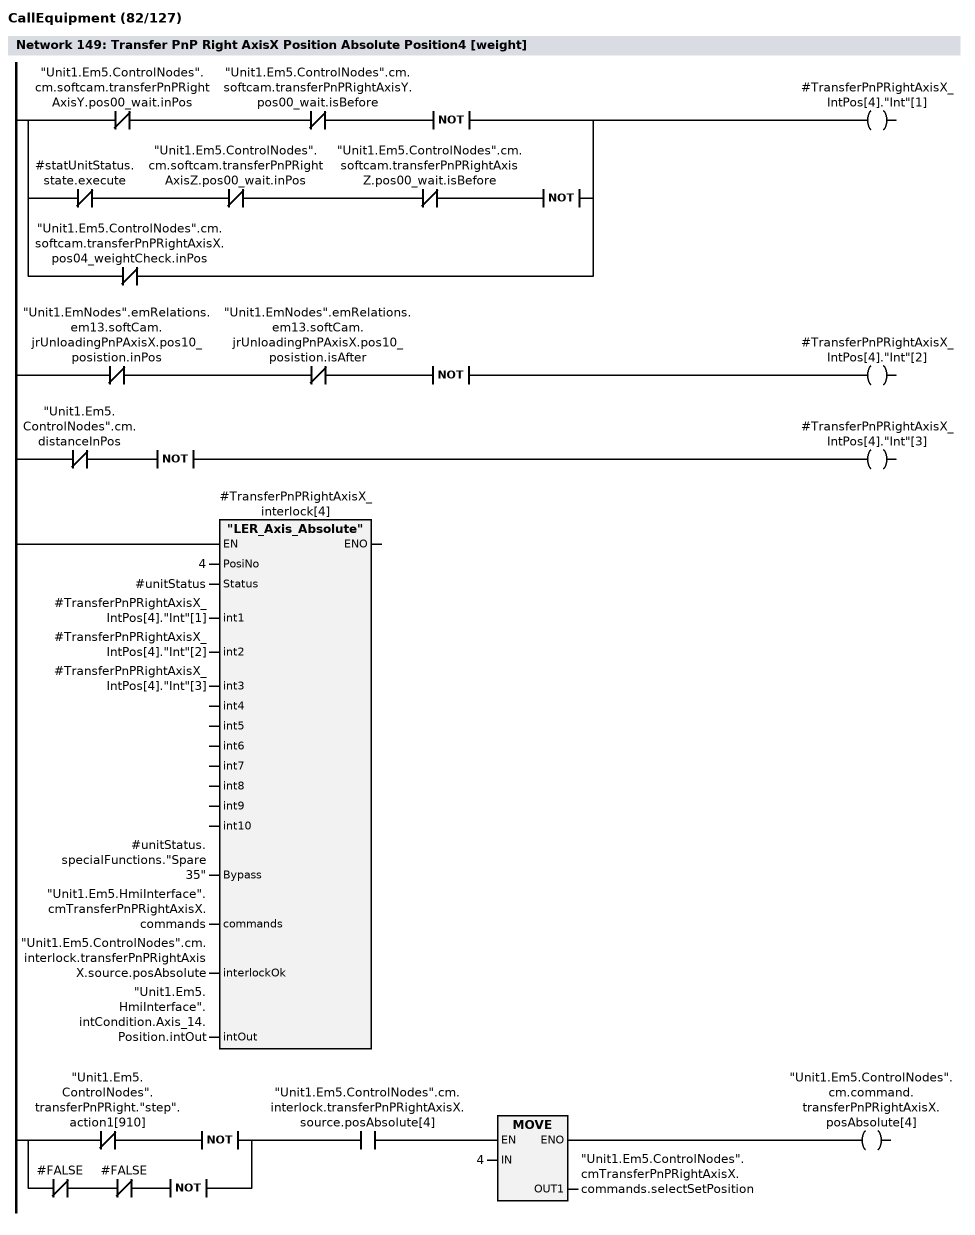
   RUNG wire#powerrail
      I_Contact( "Unit1.Em5.ControlNodes".cm.softcam.transferPnPRightAxisY.pos00_wait.inPos )
      I_Contact( "Unit1.Em5.ControlNodes".cm.softcam.transferPnPRightAxisY.pos00_wait.isBefore )
      Not()
      wire#w1
      Coil( #TransferPnPRightAxisX_IntPos[4]."Int"[1] )
   END_RUNG
   RUNG wire#powerrail
      I_Contact( #statUnitStatus.state.execute )
      I_Contact( "Unit1.Em5.ControlNodes".cm.softcam.transferPnPRightAxisZ.pos00_wait.inPos )
      I_Contact( "Unit1.Em5.ControlNodes".cm.softcam.transferPnPRightAxisZ.pos00_wait.isBefore )
      Not()
   END_RUNG wire#w1
   RUNG wire#powerrail
      I_Contact( "Unit1.Em5.ControlNodes".cm.softcam.transferPnPRightAxisX.pos04_weightCheck.inPos )
   END_RUNG wire#w1
   RUNG wire#powerrail
      I_Contact( "Unit1.EmNodes".emRelations.em13.softCam.jrUnIoadingPnPAxisX.pos10_posistion.inPos )
      I_Contact( "Unit1.EmNodes".emRelations.em13.softCam.jrUnIoadingPnPAxisX.pos10_posistion.isAfter )
      Not()
      Coil( #TransferPnPRightAxisX_IntPos[4]."Int"[2] )
   END_RUNG
   RUNG wire#powerrail
      I_Contact( "Unit1.Em5.ControlNodes".cm.distanceInPos )
      Not()
      Coil( #TransferPnPRightAxisX_IntPos[4]."Int"[3] )
   END_RUNG
   RUNG wire#powerrail
      #TransferPnPRightAxisX_interlock[4](PosiNo := 4, Status := #unitStatus, int1 := #TransferPnPRightAxisX_IntPos[4]."Int"[1], int2 := #TransferPnPRightAxisX_IntPos[4]."Int"[2], int3 := #TransferPnPRightAxisX_IntPos[4]."Int"[3], int4 :=, int5 :=, int6 :=, int7 :=, int8 :=, int9 :=, int10 :=, Bypass := #unitStatus.specialFunctions."Spare 35", commands := "Unit1.Em5.HmiInterface".cmTransferPnPRightAxisX.commands, interlockOk := "Unit1.Em5.ControlNodes".cm.interlock.transferPnPRightAxisX.source.posAbsolute, intOut := "Unit1.Em5.HmiInterface".intCondition.Axis_14.Position.intOut)
   END_RUNG
   RUNG wire#powerrail
      I_Contact( "Unit1.Em5.ControlNodes".transferPnPRight."step".action1[910] )
      Not()
      wire#w2
      Contact( "Unit1.Em5.ControlNodes".cm.interlock.transferPnPRightAxisX.source.posAbsolute[4] )
      Move(in := 4, out1 => "Unit1.Em5.ControlNodes".cmTransferPnPRightAxisX.commands.selectSetPosition)
      Coil( "Unit1.Em5.ControlNodes".cm.command.transferPnPRightAxisX.posAbsolute[4] )
   END_RUNG
   RUNG wire#powerrail
      I_Contact( #FALSE )
      I_Contact( #FALSE )
      Not()
   END_RUNG wire#w2
   // the same network as SCL:
   #TransferPnPRightAxisX_IntPos[4]."Int"[1] := NOT (NOT "Unit1.Em5.ControlNodes".cm.softcam.transferPnPRightAxisY.pos00_wait.inPos AND NOT "Unit1.Em5.ControlNodes".cm.softcam.transferPnPRightAxisY.pos00_wait.isBefore) OR NOT (NOT #statUnitStatus.state.execute AND NOT "Unit1.Em5.ControlNodes".cm.softcam.transferPnPRightAxisZ.pos00_wait.inPos AND NOT "Unit1.Em5.ControlNodes".cm.softcam.transferPnPRightAxisZ.pos00_wait.isBefore) OR NOT "Unit1.Em5.ControlNodes".cm.softcam.transferPnPRightAxisX.pos04_weightCheck.inPos;
   #TransferPnPRightAxisX_IntPos[4]."Int"[2] := NOT (NOT "Unit1.EmNodes".emRelations.em13.softCam.jrUnIoadingPnPAxisX.pos10_posistion.inPos AND NOT "Unit1.EmNodes".emRelations.em13.softCam.jrUnIoadingPnPAxisX.pos10_posistion.isAfter);
   #TransferPnPRightAxisX_IntPos[4]."Int"[3] := NOT (NOT "Unit1.Em5.ControlNodes".cm.distanceInPos);
   #TransferPnPRightAxisX_interlock[4](PosiNo := 4,   // "LER_Axis_Absolute"
                           Status := #unitStatus,
                           int1 := #TransferPnPRightAxisX_IntPos[4]."Int"[1],
                           int2 := #TransferPnPRightAxisX_IntPos[4]."Int"[2],
                           int3 := #TransferPnPRightAxisX_IntPos[4]."Int"[3],
                           Bypass := #unitStatus.specialFunctions."Spare 35",
                           commands := "Unit1.Em5.HmiInterface".cmTransferPnPRightAxisX.commands,
                           interlockOk := "Unit1.Em5.ControlNodes".cm.interlock.transferPnPRightAxisX.source.posAbsolute,
                           intOut := "Unit1.Em5.HmiInterface".intCondition.Axis_14.Position.intOut);
   #_w1 := (NOT (NOT "Unit1.Em5.ControlNodes".transferPnPRight."step".action1[910]) OR NOT (NOT #FALSE AND NOT #FALSE)) AND "Unit1.Em5.ControlNodes".cm.interlock.transferPnPRightAxisX.source.posAbsolute[4];
   IF #_w1 THEN "Unit1.Em5.ControlNodes".cmTransferPnPRightAxisX.commands.selectSetPosition := 4; END_IF;
   "Unit1.Em5.ControlNodes".cm.command.transferPnPRightAxisX.posAbsolute[4] := #_w1;
END_REGION

REGION Network 150: Transfer PnP Right AxisX Position Absolute Position5
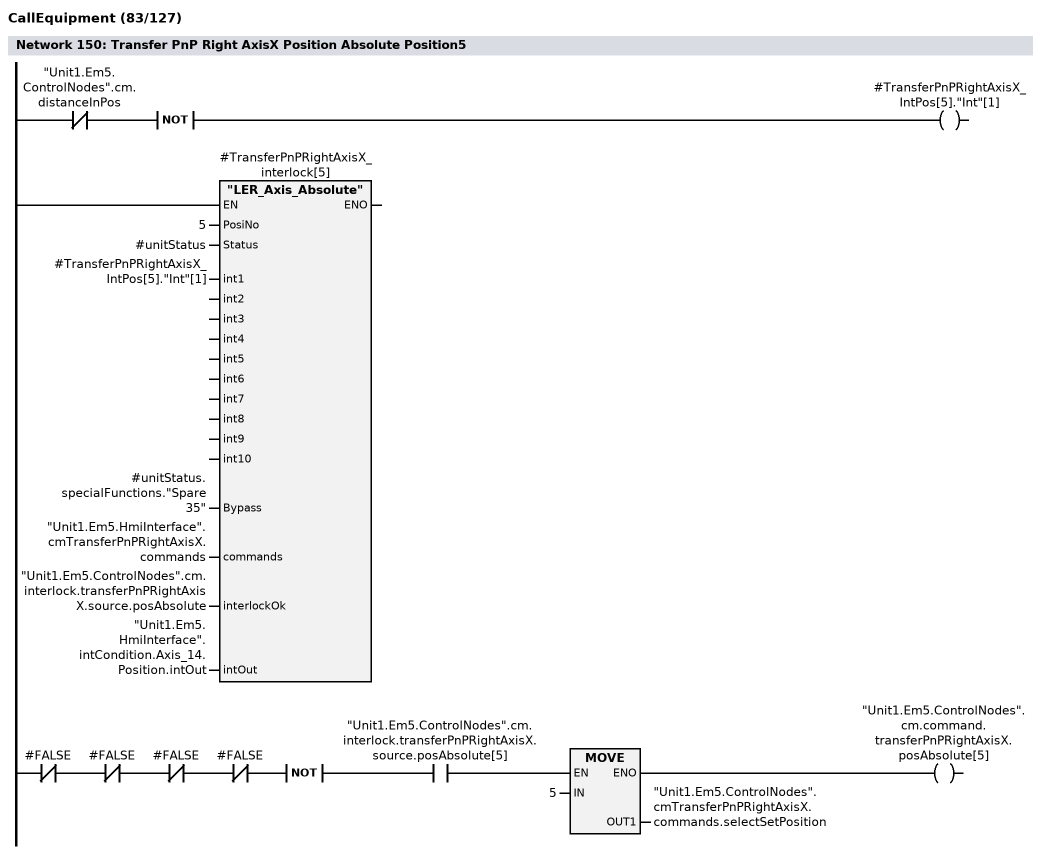
   RUNG wire#powerrail
      I_Contact( "Unit1.Em5.ControlNodes".cm.distanceInPos )
      Not()
      Coil( #TransferPnPRightAxisX_IntPos[5]."Int"[1] )
   END_RUNG
   RUNG wire#powerrail
      #TransferPnPRightAxisX_interlock[5](PosiNo := 5, Status := #unitStatus, int1 := #TransferPnPRightAxisX_IntPos[5]."Int"[1], int2 :=, int3 :=, int4 :=, int5 :=, int6 :=, int7 :=, int8 :=, int9 :=, int10 :=, Bypass := #unitStatus.specialFunctions."Spare 35", commands := "Unit1.Em5.HmiInterface".cmTransferPnPRightAxisX.commands, interlockOk := "Unit1.Em5.ControlNodes".cm.interlock.transferPnPRightAxisX.source.posAbsolute, intOut := "Unit1.Em5.HmiInterface".intCondition.Axis_14.Position.intOut)
   END_RUNG
   RUNG wire#powerrail
      I_Contact( #FALSE )
      I_Contact( #FALSE )
      I_Contact( #FALSE )
      I_Contact( #FALSE )
      Not()
      Contact( "Unit1.Em5.ControlNodes".cm.interlock.transferPnPRightAxisX.source.posAbsolute[5] )
      Move(in := 5, out1 => "Unit1.Em5.ControlNodes".cmTransferPnPRightAxisX.commands.selectSetPosition)
      Coil( "Unit1.Em5.ControlNodes".cm.command.transferPnPRightAxisX.posAbsolute[5] )
   END_RUNG
   // the same network as SCL:
   #TransferPnPRightAxisX_IntPos[5]."Int"[1] := NOT (NOT "Unit1.Em5.ControlNodes".cm.distanceInPos);
   #TransferPnPRightAxisX_interlock[5](PosiNo := 5,   // "LER_Axis_Absolute"
                           Status := #unitStatus,
                           int1 := #TransferPnPRightAxisX_IntPos[5]."Int"[1],
                           Bypass := #unitStatus.specialFunctions."Spare 35",
                           commands := "Unit1.Em5.HmiInterface".cmTransferPnPRightAxisX.commands,
                           interlockOk := "Unit1.Em5.ControlNodes".cm.interlock.transferPnPRightAxisX.source.posAbsolute,
                           intOut := "Unit1.Em5.HmiInterface".intCondition.Axis_14.Position.intOut);
   #_w1 := NOT (NOT #FALSE AND NOT #FALSE AND NOT #FALSE AND NOT #FALSE) AND "Unit1.Em5.ControlNodes".cm.interlock.transferPnPRightAxisX.source.posAbsolute[5];
   IF #_w1 THEN "Unit1.Em5.ControlNodes".cmTransferPnPRightAxisX.commands.selectSetPosition := 5; END_IF;
   "Unit1.Em5.ControlNodes".cm.command.transferPnPRightAxisX.posAbsolute[5] := #_w1;
END_REGION

REGION Network 151: Transfer PnP Right AxisX Position Absolute Position7
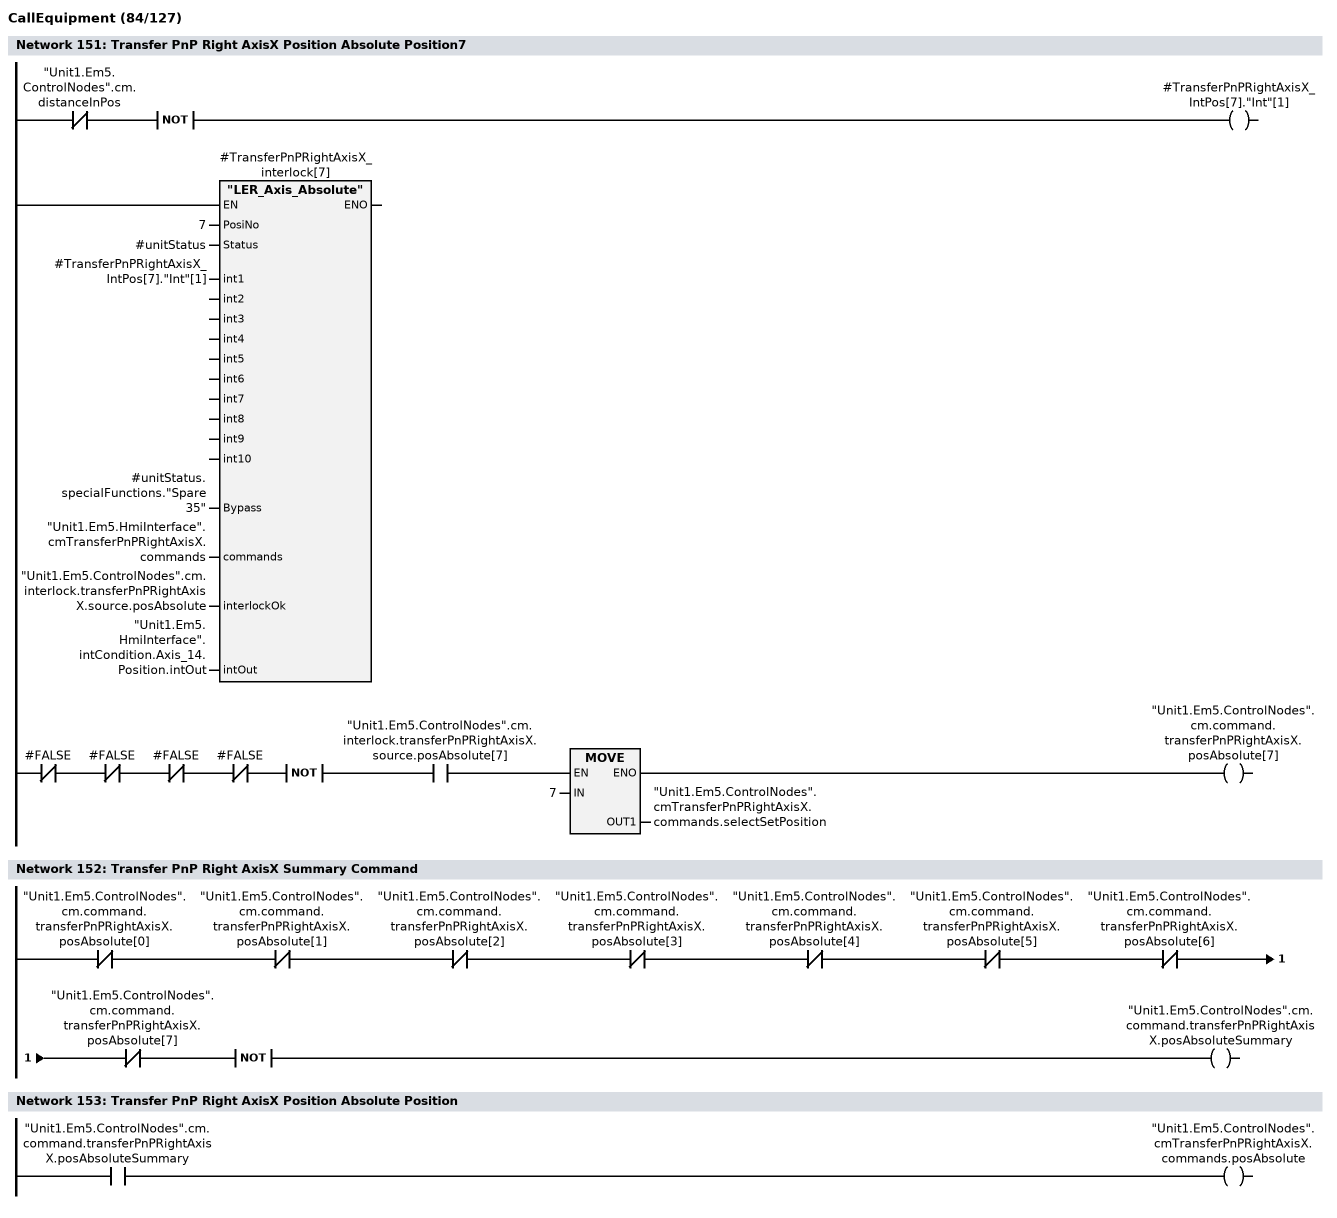
   RUNG wire#powerrail
      I_Contact( "Unit1.Em5.ControlNodes".cm.distanceInPos )
      Not()
      Coil( #TransferPnPRightAxisX_IntPos[7]."Int"[1] )
   END_RUNG
   RUNG wire#powerrail
      #TransferPnPRightAxisX_interlock[7](PosiNo := 7, Status := #unitStatus, int1 := #TransferPnPRightAxisX_IntPos[7]."Int"[1], int2 :=, int3 :=, int4 :=, int5 :=, int6 :=, int7 :=, int8 :=, int9 :=, int10 :=, Bypass := #unitStatus.specialFunctions."Spare 35", commands := "Unit1.Em5.HmiInterface".cmTransferPnPRightAxisX.commands, interlockOk := "Unit1.Em5.ControlNodes".cm.interlock.transferPnPRightAxisX.source.posAbsolute, intOut := "Unit1.Em5.HmiInterface".intCondition.Axis_14.Position.intOut)
   END_RUNG
   RUNG wire#powerrail
      I_Contact( #FALSE )
      I_Contact( #FALSE )
      I_Contact( #FALSE )
      I_Contact( #FALSE )
      Not()
      Contact( "Unit1.Em5.ControlNodes".cm.interlock.transferPnPRightAxisX.source.posAbsolute[7] )
      Move(in := 7, out1 => "Unit1.Em5.ControlNodes".cmTransferPnPRightAxisX.commands.selectSetPosition)
      Coil( "Unit1.Em5.ControlNodes".cm.command.transferPnPRightAxisX.posAbsolute[7] )
   END_RUNG
   // the same network as SCL:
   #TransferPnPRightAxisX_IntPos[7]."Int"[1] := NOT (NOT "Unit1.Em5.ControlNodes".cm.distanceInPos);
   #TransferPnPRightAxisX_interlock[7](PosiNo := 7,   // "LER_Axis_Absolute"
                           Status := #unitStatus,
                           int1 := #TransferPnPRightAxisX_IntPos[7]."Int"[1],
                           Bypass := #unitStatus.specialFunctions."Spare 35",
                           commands := "Unit1.Em5.HmiInterface".cmTransferPnPRightAxisX.commands,
                           interlockOk := "Unit1.Em5.ControlNodes".cm.interlock.transferPnPRightAxisX.source.posAbsolute,
                           intOut := "Unit1.Em5.HmiInterface".intCondition.Axis_14.Position.intOut);
   #_w1 := NOT (NOT #FALSE AND NOT #FALSE AND NOT #FALSE AND NOT #FALSE) AND "Unit1.Em5.ControlNodes".cm.interlock.transferPnPRightAxisX.source.posAbsolute[7];
   IF #_w1 THEN "Unit1.Em5.ControlNodes".cmTransferPnPRightAxisX.commands.selectSetPosition := 7; END_IF;
   "Unit1.Em5.ControlNodes".cm.command.transferPnPRightAxisX.posAbsolute[7] := #_w1;
END_REGION

REGION Network 152: Transfer PnP Right AxisX Summary Command
   RUNG wire#powerrail
      I_Contact( "Unit1.Em5.ControlNodes".cm.command.transferPnPRightAxisX.posAbsolute[0] )
      I_Contact( "Unit1.Em5.ControlNodes".cm.command.transferPnPRightAxisX.posAbsolute[1] )
      I_Contact( "Unit1.Em5.ControlNodes".cm.command.transferPnPRightAxisX.posAbsolute[2] )
      I_Contact( "Unit1.Em5.ControlNodes".cm.command.transferPnPRightAxisX.posAbsolute[3] )
      I_Contact( "Unit1.Em5.ControlNodes".cm.command.transferPnPRightAxisX.posAbsolute[4] )
      I_Contact( "Unit1.Em5.ControlNodes".cm.command.transferPnPRightAxisX.posAbsolute[5] )
      I_Contact( "Unit1.Em5.ControlNodes".cm.command.transferPnPRightAxisX.posAbsolute[6] )
      I_Contact( "Unit1.Em5.ControlNodes".cm.command.transferPnPRightAxisX.posAbsolute[7] )
      Not()
      Coil( "Unit1.Em5.ControlNodes".cm.command.transferPnPRightAxisX.posAbsoluteSummary )
   END_RUNG
   // the same network as SCL:
   "Unit1.Em5.ControlNodes".cm.command.transferPnPRightAxisX.posAbsoluteSummary := NOT (NOT "Unit1.Em5.ControlNodes".cm.command.transferPnPRightAxisX.posAbsolute[0] AND NOT "Unit1.Em5.ControlNodes".cm.command.transferPnPRightAxisX.posAbsolute[1] AND NOT "Unit1.Em5.ControlNodes".cm.command.transferPnPRightAxisX.posAbsolute[2] AND NOT "Unit1.Em5.ControlNodes".cm.command.transferPnPRightAxisX.posAbsolute[3] AND NOT "Unit1.Em5.ControlNodes".cm.command.transferPnPRightAxisX.posAbsolute[4] AND NOT "Unit1.Em5.ControlNodes".cm.command.transferPnPRightAxisX.posAbsolute[5] AND NOT "Unit1.Em5.ControlNodes".cm.command.transferPnPRightAxisX.posAbsolute[6] AND NOT "Unit1.Em5.ControlNodes".cm.command.transferPnPRightAxisX.posAbsolute[7]);
END_REGION

REGION Network 153: Transfer PnP Right AxisX Position Absolute Position
   RUNG wire#powerrail
      Contact( "Unit1.Em5.ControlNodes".cm.command.transferPnPRightAxisX.posAbsoluteSummary )
      Coil( "Unit1.Em5.ControlNodes".cmTransferPnPRightAxisX.commands.posAbsolute )
   END_RUNG
   // the same network as SCL:
   "Unit1.Em5.ControlNodes".cmTransferPnPRightAxisX.commands.posAbsolute := "Unit1.Em5.ControlNodes".cm.command.transferPnPRightAxisX.posAbsoluteSummary;
END_REGION

REGION Network 154: Transfer PnP Right AxisX Interlock Summary
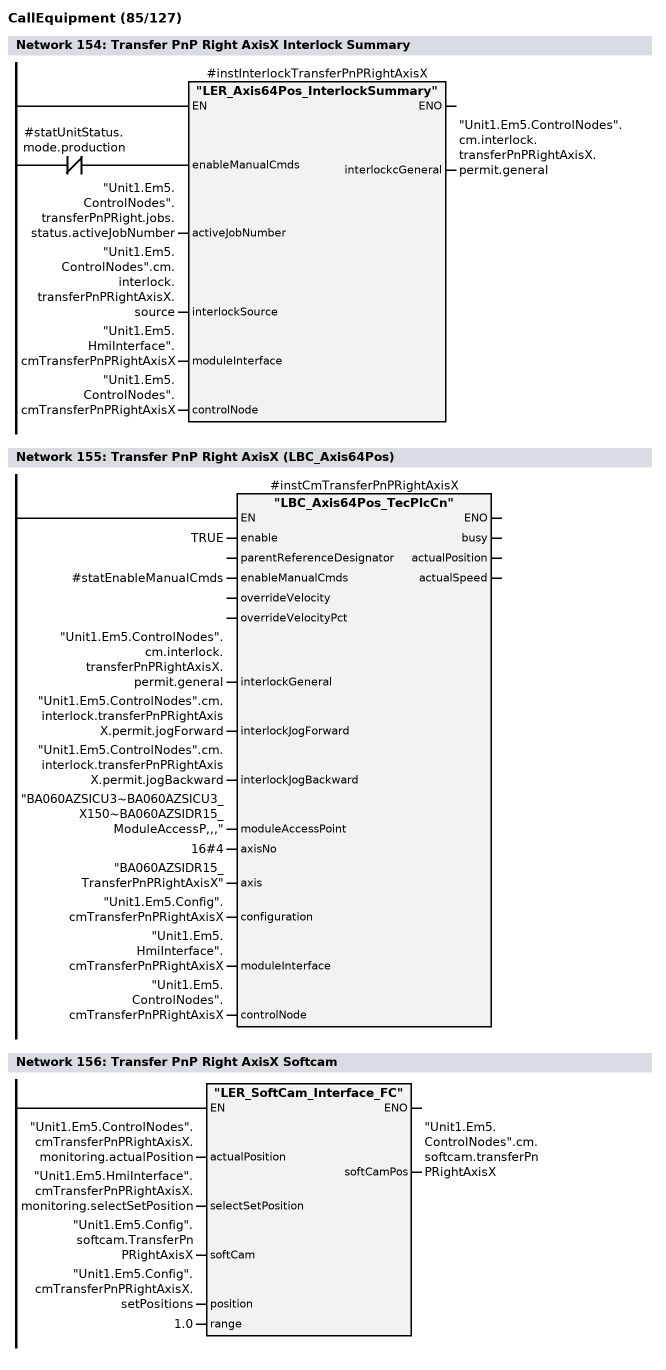
   RUNG wire#powerrail
      #instInterlockTransferPnPRightAxisX(enableManualCmds := wire#w1, activeJobNumber := "Unit1.Em5.ControlNodes".transferPnPRight.jobs.status.activeJobNumber, interlockSource := "Unit1.Em5.ControlNodes".cm.interlock.transferPnPRightAxisX.source, moduleInterface := "Unit1.Em5.HmiInterface".cmTransferPnPRightAxisX, controlNode := "Unit1.Em5.ControlNodes".cmTransferPnPRightAxisX, interlockcGeneral => "Unit1.Em5.ControlNodes".cm.interlock.transferPnPRightAxisX.permit.general)
   END_RUNG
   RUNG wire#powerrail
      I_Contact( #statUnitStatus.mode.production )
   END_RUNG wire#w1
   // the same network as SCL:
   #instInterlockTransferPnPRightAxisX(enableManualCmds := NOT #statUnitStatus.mode.production,   // "LER_Axis64Pos_InterlockSummary"
                           activeJobNumber := "Unit1.Em5.ControlNodes".transferPnPRight.jobs.status.activeJobNumber,
                           interlockSource := "Unit1.Em5.ControlNodes".cm.interlock.transferPnPRightAxisX.source,
                           moduleInterface := "Unit1.Em5.HmiInterface".cmTransferPnPRightAxisX,
                           controlNode := "Unit1.Em5.ControlNodes".cmTransferPnPRightAxisX,
                           interlockcGeneral => "Unit1.Em5.ControlNodes".cm.interlock.transferPnPRightAxisX.permit.general);
END_REGION

REGION Network 155: Transfer PnP Right AxisX (LBC_Axis64Pos)
   RUNG wire#powerrail
      #instCmTransferPnPRightAxisX(enable := TRUE, parentReferenceDesignator :=, enableManualCmds := #statEnableManualCmds, overrideVelocity :=, overrideVelocityPct :=, interlockGeneral := "Unit1.Em5.ControlNodes".cm.interlock.transferPnPRightAxisX.permit.general, interlockJogForward := "Unit1.Em5.ControlNodes".cm.interlock.transferPnPRightAxisX.permit.jogForward, interlockJogBackward := "Unit1.Em5.ControlNodes".cm.interlock.transferPnPRightAxisX.permit.jogBackward, moduleAccessPoint := "BA060AZSICU3~BA060AZSICU3_X150~BA060AZSIDR15_ModuleAccessP,,,", axisNo := 16#4, axis := "BA060AZSIDR15_TransferPnPRightAxisX", configuration := "Unit1.Em5.Config".cmTransferPnPRightAxisX, moduleInterface := "Unit1.Em5.HmiInterface".cmTransferPnPRightAxisX, controlNode := "Unit1.Em5.ControlNodes".cmTransferPnPRightAxisX, busy =>, actualPosition =>, actualSpeed =>)
   END_RUNG
   // the same network as SCL:
   #instCmTransferPnPRightAxisX(enable := TRUE,   // "LBC_Axis64Pos_TecPlcCn"
                           enableManualCmds := #statEnableManualCmds,
                           interlockGeneral := "Unit1.Em5.ControlNodes".cm.interlock.transferPnPRightAxisX.permit.general,
                           interlockJogForward := "Unit1.Em5.ControlNodes".cm.interlock.transferPnPRightAxisX.permit.jogForward,
                           interlockJogBackward := "Unit1.Em5.ControlNodes".cm.interlock.transferPnPRightAxisX.permit.jogBackward,
                           moduleAccessPoint := "BA060AZSICU3~BA060AZSICU3_X150~BA060AZSIDR15_ModuleAccessP,,,",
                           axisNo := 16#4,
                           axis := "BA060AZSIDR15_TransferPnPRightAxisX",
                           configuration := "Unit1.Em5.Config".cmTransferPnPRightAxisX,
                           moduleInterface := "Unit1.Em5.HmiInterface".cmTransferPnPRightAxisX,
                           controlNode := "Unit1.Em5.ControlNodes".cmTransferPnPRightAxisX);
END_REGION

REGION Network 156: Transfer PnP Right AxisX Softcam
   RUNG wire#powerrail
      "LER_SoftCam_Interface_FC"(actualPosition := "Unit1.Em5.ControlNodes".cmTransferPnPRightAxisX.monitoring.actualPosition, selectSetPosition := "Unit1.Em5.HmiInterface".cmTransferPnPRightAxisX.monitoring.selectSetPosition, softCam := "Unit1.Em5.Config".softcam.TransferPnPRightAxisX, position := "Unit1.Em5.Config".cmTransferPnPRightAxisX.setPositions, range := 1.0, softCamPos => "Unit1.Em5.ControlNodes".cm.softcam.transferPnPRightAxisX)
   END_RUNG
   // the same network as SCL:
   "LER_SoftCam_Interface_FC"(actualPosition := "Unit1.Em5.ControlNodes".cmTransferPnPRightAxisX.monitoring.actualPosition,
                           selectSetPosition := "Unit1.Em5.HmiInterface".cmTransferPnPRightAxisX.monitoring.selectSetPosition,
                           softCam := "Unit1.Em5.Config".softcam.TransferPnPRightAxisX,
                           position := "Unit1.Em5.Config".cmTransferPnPRightAxisX.setPositions,
                           range := 1.0,
                           softCamPos => "Unit1.Em5.ControlNodes".cm.softcam.transferPnPRightAxisX);
END_REGION

REGION Network 158: Transfer P&P Right Y-Axis Upload Actual Current And Torque Values
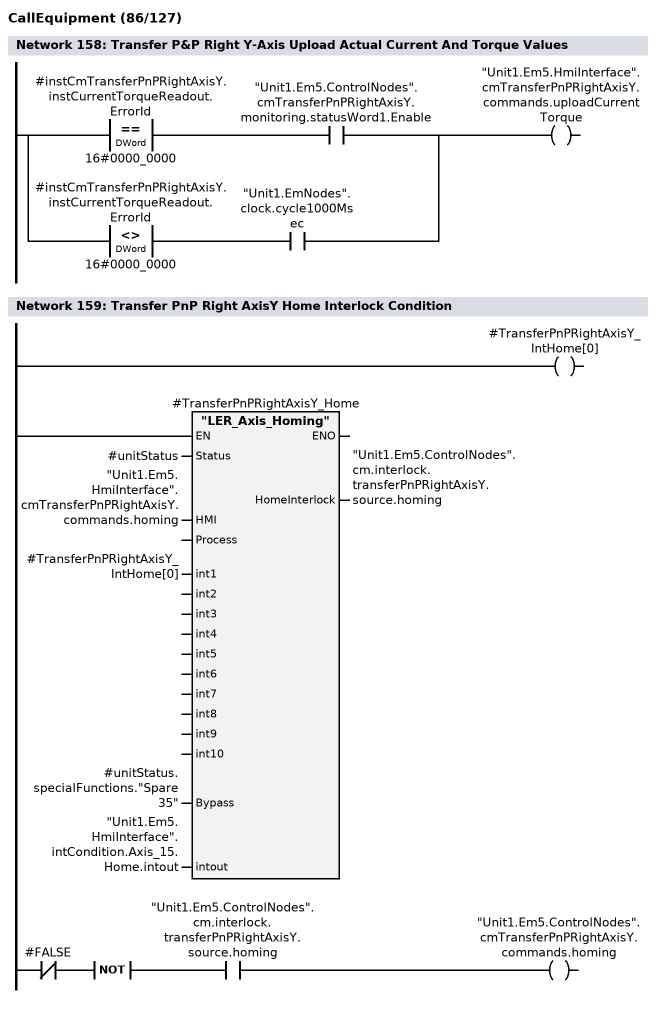
   RUNG wire#powerrail
      { S7_Templates := "SrcType := DWord" } EQ_Contact(in1 := #instCmTransferPnPRightAxisY.instCurrentTorqueReadout.ErrorId, in2 := 16#0000_0000)
      Contact( "Unit1.Em5.ControlNodes".cmTransferPnPRightAxisY.monitoring.statusWord1.Enable )
      wire#w1
      Coil( "Unit1.Em5.HmiInterface".cmTransferPnPRightAxisY.commands.uploadCurrentTorque )
   END_RUNG
   RUNG wire#powerrail
      { S7_Templates := "SrcType := DWord" } NE_Contact(in1 := #instCmTransferPnPRightAxisY.instCurrentTorqueReadout.ErrorId, in2 := 16#0000_0000)
      Contact( "Unit1.EmNodes".clock.cycle1000Msec )
   END_RUNG wire#w1
   // the same network as SCL:
   "Unit1.Em5.HmiInterface".cmTransferPnPRightAxisY.commands.uploadCurrentTorque := ((#instCmTransferPnPRightAxisY.instCurrentTorqueReadout.ErrorId = 16#0000_0000) AND "Unit1.Em5.ControlNodes".cmTransferPnPRightAxisY.monitoring.statusWord1.Enable) OR ((#instCmTransferPnPRightAxisY.instCurrentTorqueReadout.ErrorId <> 16#0000_0000) AND "Unit1.EmNodes".clock.cycle1000Msec);
END_REGION

REGION Network 159: Transfer PnP Right AxisY Home Interlock Condition
   RUNG wire#powerrail
      Coil( #TransferPnPRightAxisY_IntHome[0] )
   END_RUNG
   RUNG wire#powerrail
      #TransferPnPRightAxisY_Home(Status := #unitStatus, HMI := "Unit1.Em5.HmiInterface".cmTransferPnPRightAxisY.commands.homing, Process :=, int1 := #TransferPnPRightAxisY_IntHome[0], int2 :=, int3 :=, int4 :=, int5 :=, int6 :=, int7 :=, int8 :=, int9 :=, int10 :=, Bypass := #unitStatus.specialFunctions."Spare 35", intout := "Unit1.Em5.HmiInterface".intCondition.Axis_15.Home.intout, HomeInterlock => "Unit1.Em5.ControlNodes".cm.interlock.transferPnPRightAxisY.source.homing)
   END_RUNG
   RUNG wire#powerrail
      I_Contact( #FALSE )
      Not()
      Contact( "Unit1.Em5.ControlNodes".cm.interlock.transferPnPRightAxisY.source.homing )
      Coil( "Unit1.Em5.ControlNodes".cmTransferPnPRightAxisY.commands.homing )
   END_RUNG
   // the same network as SCL:
   #TransferPnPRightAxisY_IntHome[0] := TRUE;
   #TransferPnPRightAxisY_Home(Status := #unitStatus,   // "LER_Axis_Homing"
                           HMI := "Unit1.Em5.HmiInterface".cmTransferPnPRightAxisY.commands.homing,
                           int1 := #TransferPnPRightAxisY_IntHome[0],
                           Bypass := #unitStatus.specialFunctions."Spare 35",
                           intout := "Unit1.Em5.HmiInterface".intCondition.Axis_15.Home.intout,
                           HomeInterlock => "Unit1.Em5.ControlNodes".cm.interlock.transferPnPRightAxisY.source.homing);
   "Unit1.Em5.ControlNodes".cmTransferPnPRightAxisY.commands.homing := NOT (NOT #FALSE) AND "Unit1.Em5.ControlNodes".cm.interlock.transferPnPRightAxisY.source.homing;
END_REGION

REGION Network 160: Transfer PnP Right AxisY JOG Interlock Condition
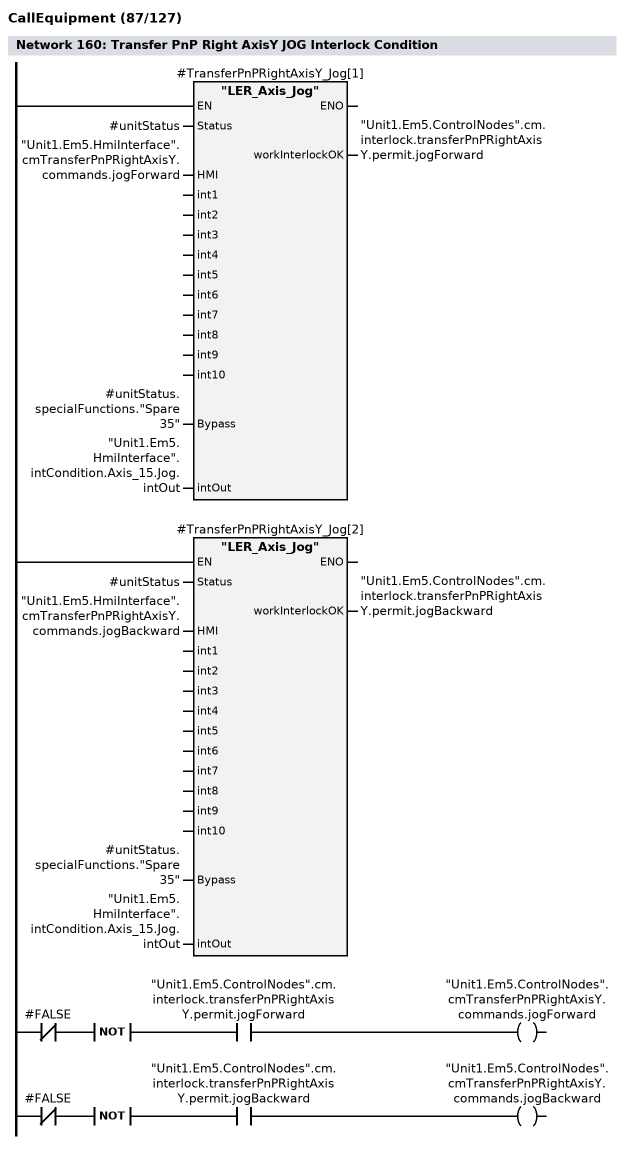
   RUNG wire#powerrail
      #TransferPnPRightAxisY_Jog[1](Status := #unitStatus, HMI := "Unit1.Em5.HmiInterface".cmTransferPnPRightAxisY.commands.jogForward, int1 :=, int2 :=, int3 :=, int4 :=, int5 :=, int6 :=, int7 :=, int8 :=, int9 :=, int10 :=, Bypass := #unitStatus.specialFunctions."Spare 35", intOut := "Unit1.Em5.HmiInterface".intCondition.Axis_15.Jog.intOut, workInterlockOK => "Unit1.Em5.ControlNodes".cm.interlock.transferPnPRightAxisY.permit.jogForward)
   END_RUNG
   RUNG wire#powerrail
      #TransferPnPRightAxisY_Jog[2](Status := #unitStatus, HMI := "Unit1.Em5.HmiInterface".cmTransferPnPRightAxisY.commands.jogBackward, int1 :=, int2 :=, int3 :=, int4 :=, int5 :=, int6 :=, int7 :=, int8 :=, int9 :=, int10 :=, Bypass := #unitStatus.specialFunctions."Spare 35", intOut := "Unit1.Em5.HmiInterface".intCondition.Axis_15.Jog.intOut, workInterlockOK => "Unit1.Em5.ControlNodes".cm.interlock.transferPnPRightAxisY.permit.jogBackward)
   END_RUNG
   RUNG wire#powerrail
      I_Contact( #FALSE )
      Not()
      Contact( "Unit1.Em5.ControlNodes".cm.interlock.transferPnPRightAxisY.permit.jogForward )
      Coil( "Unit1.Em5.ControlNodes".cmTransferPnPRightAxisY.commands.jogForward )
   END_RUNG
   RUNG wire#powerrail
      I_Contact( #FALSE )
      Not()
      Contact( "Unit1.Em5.ControlNodes".cm.interlock.transferPnPRightAxisY.permit.jogBackward )
      Coil( "Unit1.Em5.ControlNodes".cmTransferPnPRightAxisY.commands.jogBackward )
   END_RUNG
   // the same network as SCL:
   #TransferPnPRightAxisY_Jog[1](Status := #unitStatus,   // "LER_Axis_Jog"
                           HMI := "Unit1.Em5.HmiInterface".cmTransferPnPRightAxisY.commands.jogForward,
                           Bypass := #unitStatus.specialFunctions."Spare 35",
                           intOut := "Unit1.Em5.HmiInterface".intCondition.Axis_15.Jog.intOut,
                           workInterlockOK => "Unit1.Em5.ControlNodes".cm.interlock.transferPnPRightAxisY.permit.jogForward);
   #TransferPnPRightAxisY_Jog[2](Status := #unitStatus,   // "LER_Axis_Jog"
                           HMI := "Unit1.Em5.HmiInterface".cmTransferPnPRightAxisY.commands.jogBackward,
                           Bypass := #unitStatus.specialFunctions."Spare 35",
                           intOut := "Unit1.Em5.HmiInterface".intCondition.Axis_15.Jog.intOut,
                           workInterlockOK => "Unit1.Em5.ControlNodes".cm.interlock.transferPnPRightAxisY.permit.jogBackward);
   "Unit1.Em5.ControlNodes".cmTransferPnPRightAxisY.commands.jogForward := NOT (NOT #FALSE) AND "Unit1.Em5.ControlNodes".cm.interlock.transferPnPRightAxisY.permit.jogForward;
   "Unit1.Em5.ControlNodes".cmTransferPnPRightAxisY.commands.jogBackward := NOT (NOT #FALSE) AND "Unit1.Em5.ControlNodes".cm.interlock.transferPnPRightAxisY.permit.jogBackward;
END_REGION

REGION Network 161: Transfer PnP Right AxisY Position Absolute Position0
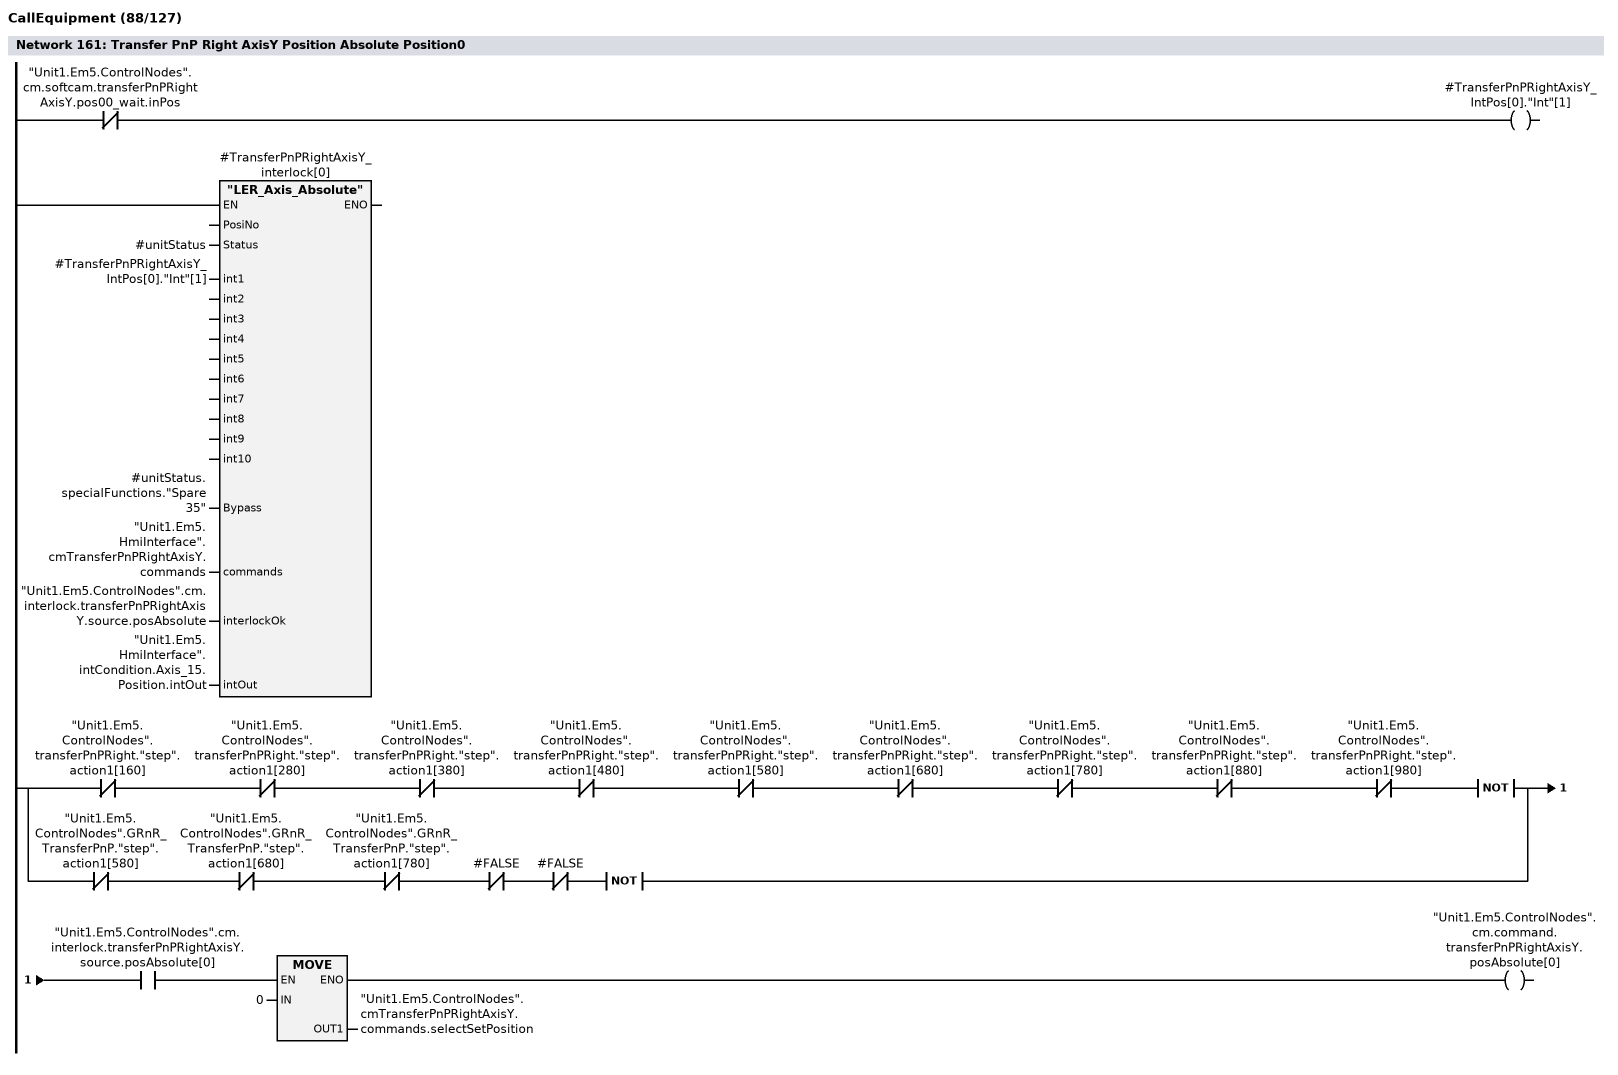
   RUNG wire#powerrail
      I_Contact( "Unit1.Em5.ControlNodes".cm.softcam.transferPnPRightAxisY.pos00_wait.inPos )
      Coil( #TransferPnPRightAxisY_IntPos[0]."Int"[1] )
   END_RUNG
   RUNG wire#powerrail
      #TransferPnPRightAxisY_interlock[0](PosiNo :=, Status := #unitStatus, int1 := #TransferPnPRightAxisY_IntPos[0]."Int"[1], int2 :=, int3 :=, int4 :=, int5 :=, int6 :=, int7 :=, int8 :=, int9 :=, int10 :=, Bypass := #unitStatus.specialFunctions."Spare 35", commands := "Unit1.Em5.HmiInterface".cmTransferPnPRightAxisY.commands, interlockOk := "Unit1.Em5.ControlNodes".cm.interlock.transferPnPRightAxisY.source.posAbsolute, intOut := "Unit1.Em5.HmiInterface".intCondition.Axis_15.Position.intOut)
   END_RUNG
   RUNG wire#powerrail
      I_Contact( "Unit1.Em5.ControlNodes".transferPnPRight."step".action1[160] )
      I_Contact( "Unit1.Em5.ControlNodes".transferPnPRight."step".action1[280] )
      I_Contact( "Unit1.Em5.ControlNodes".transferPnPRight."step".action1[380] )
      I_Contact( "Unit1.Em5.ControlNodes".transferPnPRight."step".action1[480] )
      I_Contact( "Unit1.Em5.ControlNodes".transferPnPRight."step".action1[580] )
      I_Contact( "Unit1.Em5.ControlNodes".transferPnPRight."step".action1[680] )
      I_Contact( "Unit1.Em5.ControlNodes".transferPnPRight."step".action1[780] )
      I_Contact( "Unit1.Em5.ControlNodes".transferPnPRight."step".action1[880] )
      I_Contact( "Unit1.Em5.ControlNodes".transferPnPRight."step".action1[980] )
      Not()
      wire#w1
      Contact( "Unit1.Em5.ControlNodes".cm.interlock.transferPnPRightAxisY.source.posAbsolute[0] )
      Move(in := 0, out1 => "Unit1.Em5.ControlNodes".cmTransferPnPRightAxisY.commands.selectSetPosition)
      Coil( "Unit1.Em5.ControlNodes".cm.command.transferPnPRightAxisY.posAbsolute[0] )
   END_RUNG
   RUNG wire#powerrail
      I_Contact( "Unit1.Em5.ControlNodes".GRnR_TransferPnP."step".action1[580] )
      I_Contact( "Unit1.Em5.ControlNodes".GRnR_TransferPnP."step".action1[680] )
      I_Contact( "Unit1.Em5.ControlNodes".GRnR_TransferPnP."step".action1[780] )
      I_Contact( #FALSE )
      I_Contact( #FALSE )
      Not()
   END_RUNG wire#w1
   // the same network as SCL:
   #TransferPnPRightAxisY_IntPos[0]."Int"[1] := NOT "Unit1.Em5.ControlNodes".cm.softcam.transferPnPRightAxisY.pos00_wait.inPos;
   #TransferPnPRightAxisY_interlock[0](Status := #unitStatus,   // "LER_Axis_Absolute"
                           int1 := #TransferPnPRightAxisY_IntPos[0]."Int"[1],
                           Bypass := #unitStatus.specialFunctions."Spare 35",
                           commands := "Unit1.Em5.HmiInterface".cmTransferPnPRightAxisY.commands,
                           interlockOk := "Unit1.Em5.ControlNodes".cm.interlock.transferPnPRightAxisY.source.posAbsolute,
                           intOut := "Unit1.Em5.HmiInterface".intCondition.Axis_15.Position.intOut);
   #_w1 := (NOT (NOT "Unit1.Em5.ControlNodes".transferPnPRight."step".action1[160] AND NOT "Unit1.Em5.ControlNodes".transferPnPRight."step".action1[280] AND NOT "Unit1.Em5.ControlNodes".transferPnPRight."step".action1[380] AND NOT "Unit1.Em5.ControlNodes".transferPnPRight."step".action1[480] AND NOT "Unit1.Em5.ControlNodes".transferPnPRight."step".action1[580] AND NOT "Unit1.Em5.ControlNodes".transferPnPRight."step".action1[680] AND NOT "Unit1.Em5.ControlNodes".transferPnPRight."step".action1[780] AND NOT "Unit1.Em5.ControlNodes".transferPnPRight."step".action1[880] AND NOT "Unit1.Em5.ControlNodes".transferPnPRight."step".action1[980]) OR NOT (NOT "Unit1.Em5.ControlNodes".GRnR_TransferPnP."step".action1[580] AND NOT "Unit1.Em5.ControlNodes".GRnR_TransferPnP."step".action1[680] AND NOT "Unit1.Em5.ControlNodes".GRnR_TransferPnP."step".action1[780] AND NOT #FALSE AND NOT #FALSE)) AND "Unit1.Em5.ControlNodes".cm.interlock.transferPnPRightAxisY.source.posAbsolute[0];
   IF #_w1 THEN "Unit1.Em5.ControlNodes".cmTransferPnPRightAxisY.commands.selectSetPosition := 0; END_IF;
   "Unit1.Em5.ControlNodes".cm.command.transferPnPRightAxisY.posAbsolute[0] := #_w1;
END_REGION

REGION Network 162: Transfer PnP Right AxisY Position Absolute Position1
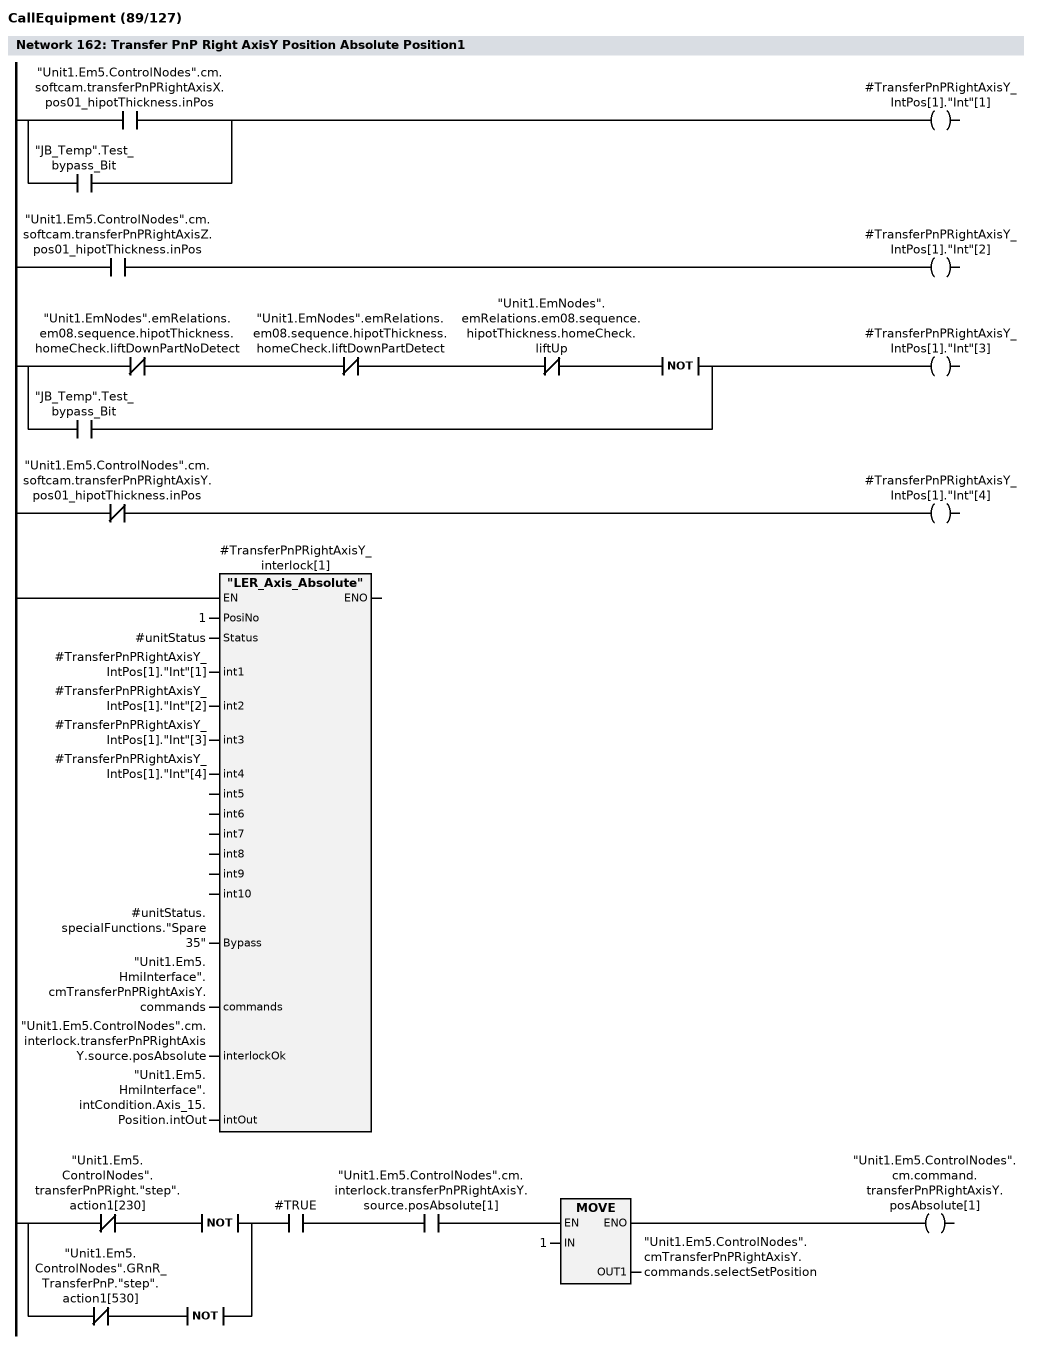
   RUNG wire#powerrail
      Contact( "Unit1.Em5.ControlNodes".cm.softcam.transferPnPRightAxisX.pos01_hipotThickness.inPos )
      wire#w1
      Coil( #TransferPnPRightAxisY_IntPos[1]."Int"[1] )
   END_RUNG
   RUNG wire#powerrail
      Contact( "JB_Temp".Test_bypass_Bit )
   END_RUNG wire#w1
   RUNG wire#powerrail
      Contact( "Unit1.Em5.ControlNodes".cm.softcam.transferPnPRightAxisZ.pos01_hipotThickness.inPos )
      Coil( #TransferPnPRightAxisY_IntPos[1]."Int"[2] )
   END_RUNG
   RUNG wire#powerrail
      I_Contact( "Unit1.EmNodes".emRelations.em08.sequence.hipotThickness.homeCheck.liftDownPartNoDetect )
      I_Contact( "Unit1.EmNodes".emRelations.em08.sequence.hipotThickness.homeCheck.liftDownPartDetect )
      I_Contact( "Unit1.EmNodes".emRelations.em08.sequence.hipotThickness.homeCheck.liftUp )
      Not()
      wire#w2
      Coil( #TransferPnPRightAxisY_IntPos[1]."Int"[3] )
   END_RUNG
   RUNG wire#powerrail
      Contact( "JB_Temp".Test_bypass_Bit )
   END_RUNG wire#w2
   RUNG wire#powerrail
      I_Contact( "Unit1.Em5.ControlNodes".cm.softcam.transferPnPRightAxisY.pos01_hipotThickness.inPos )
      Coil( #TransferPnPRightAxisY_IntPos[1]."Int"[4] )
   END_RUNG
   RUNG wire#powerrail
      #TransferPnPRightAxisY_interlock[1](PosiNo := 1, Status := #unitStatus, int1 := #TransferPnPRightAxisY_IntPos[1]."Int"[1], int2 := #TransferPnPRightAxisY_IntPos[1]."Int"[2], int3 := #TransferPnPRightAxisY_IntPos[1]."Int"[3], int4 := #TransferPnPRightAxisY_IntPos[1]."Int"[4], int5 :=, int6 :=, int7 :=, int8 :=, int9 :=, int10 :=, Bypass := #unitStatus.specialFunctions."Spare 35", commands := "Unit1.Em5.HmiInterface".cmTransferPnPRightAxisY.commands, interlockOk := "Unit1.Em5.ControlNodes".cm.interlock.transferPnPRightAxisY.source.posAbsolute, intOut := "Unit1.Em5.HmiInterface".intCondition.Axis_15.Position.intOut)
   END_RUNG
   RUNG wire#powerrail
      I_Contact( "Unit1.Em5.ControlNodes".transferPnPRight."step".action1[230] )
      Not()
      wire#w3
      Contact( #TRUE )
      Contact( "Unit1.Em5.ControlNodes".cm.interlock.transferPnPRightAxisY.source.posAbsolute[1] )
      Move(in := 1, out1 => "Unit1.Em5.ControlNodes".cmTransferPnPRightAxisY.commands.selectSetPosition)
      Coil( "Unit1.Em5.ControlNodes".cm.command.transferPnPRightAxisY.posAbsolute[1] )
   END_RUNG
   RUNG wire#powerrail
      I_Contact( "Unit1.Em5.ControlNodes".GRnR_TransferPnP."step".action1[530] )
      Not()
   END_RUNG wire#w3
   // the same network as SCL:
   #TransferPnPRightAxisY_IntPos[1]."Int"[1] := "Unit1.Em5.ControlNodes".cm.softcam.transferPnPRightAxisX.pos01_hipotThickness.inPos OR "JB_Temp".Test_bypass_Bit;
   #TransferPnPRightAxisY_IntPos[1]."Int"[2] := "Unit1.Em5.ControlNodes".cm.softcam.transferPnPRightAxisZ.pos01_hipotThickness.inPos;
   #TransferPnPRightAxisY_IntPos[1]."Int"[3] := NOT (NOT "Unit1.EmNodes".emRelations.em08.sequence.hipotThickness.homeCheck.liftDownPartNoDetect AND NOT "Unit1.EmNodes".emRelations.em08.sequence.hipotThickness.homeCheck.liftDownPartDetect AND NOT "Unit1.EmNodes".emRelations.em08.sequence.hipotThickness.homeCheck.liftUp) OR "JB_Temp".Test_bypass_Bit;
   #TransferPnPRightAxisY_IntPos[1]."Int"[4] := NOT "Unit1.Em5.ControlNodes".cm.softcam.transferPnPRightAxisY.pos01_hipotThickness.inPos;
   #TransferPnPRightAxisY_interlock[1](PosiNo := 1,   // "LER_Axis_Absolute"
                           Status := #unitStatus,
                           int1 := #TransferPnPRightAxisY_IntPos[1]."Int"[1],
                           int2 := #TransferPnPRightAxisY_IntPos[1]."Int"[2],
                           int3 := #TransferPnPRightAxisY_IntPos[1]."Int"[3],
                           int4 := #TransferPnPRightAxisY_IntPos[1]."Int"[4],
                           Bypass := #unitStatus.specialFunctions."Spare 35",
                           commands := "Unit1.Em5.HmiInterface".cmTransferPnPRightAxisY.commands,
                           interlockOk := "Unit1.Em5.ControlNodes".cm.interlock.transferPnPRightAxisY.source.posAbsolute,
                           intOut := "Unit1.Em5.HmiInterface".intCondition.Axis_15.Position.intOut);
   #_w1 := (NOT (NOT "Unit1.Em5.ControlNodes".transferPnPRight."step".action1[230]) OR NOT (NOT "Unit1.Em5.ControlNodes".GRnR_TransferPnP."step".action1[530])) AND #TRUE AND "Unit1.Em5.ControlNodes".cm.interlock.transferPnPRightAxisY.source.posAbsolute[1];
   IF #_w1 THEN "Unit1.Em5.ControlNodes".cmTransferPnPRightAxisY.commands.selectSetPosition := 1; END_IF;
   "Unit1.Em5.ControlNodes".cm.command.transferPnPRightAxisY.posAbsolute[1] := #_w1;
END_REGION

REGION Network 163: Transfer PnP Right AxisY Position Absolute Position2
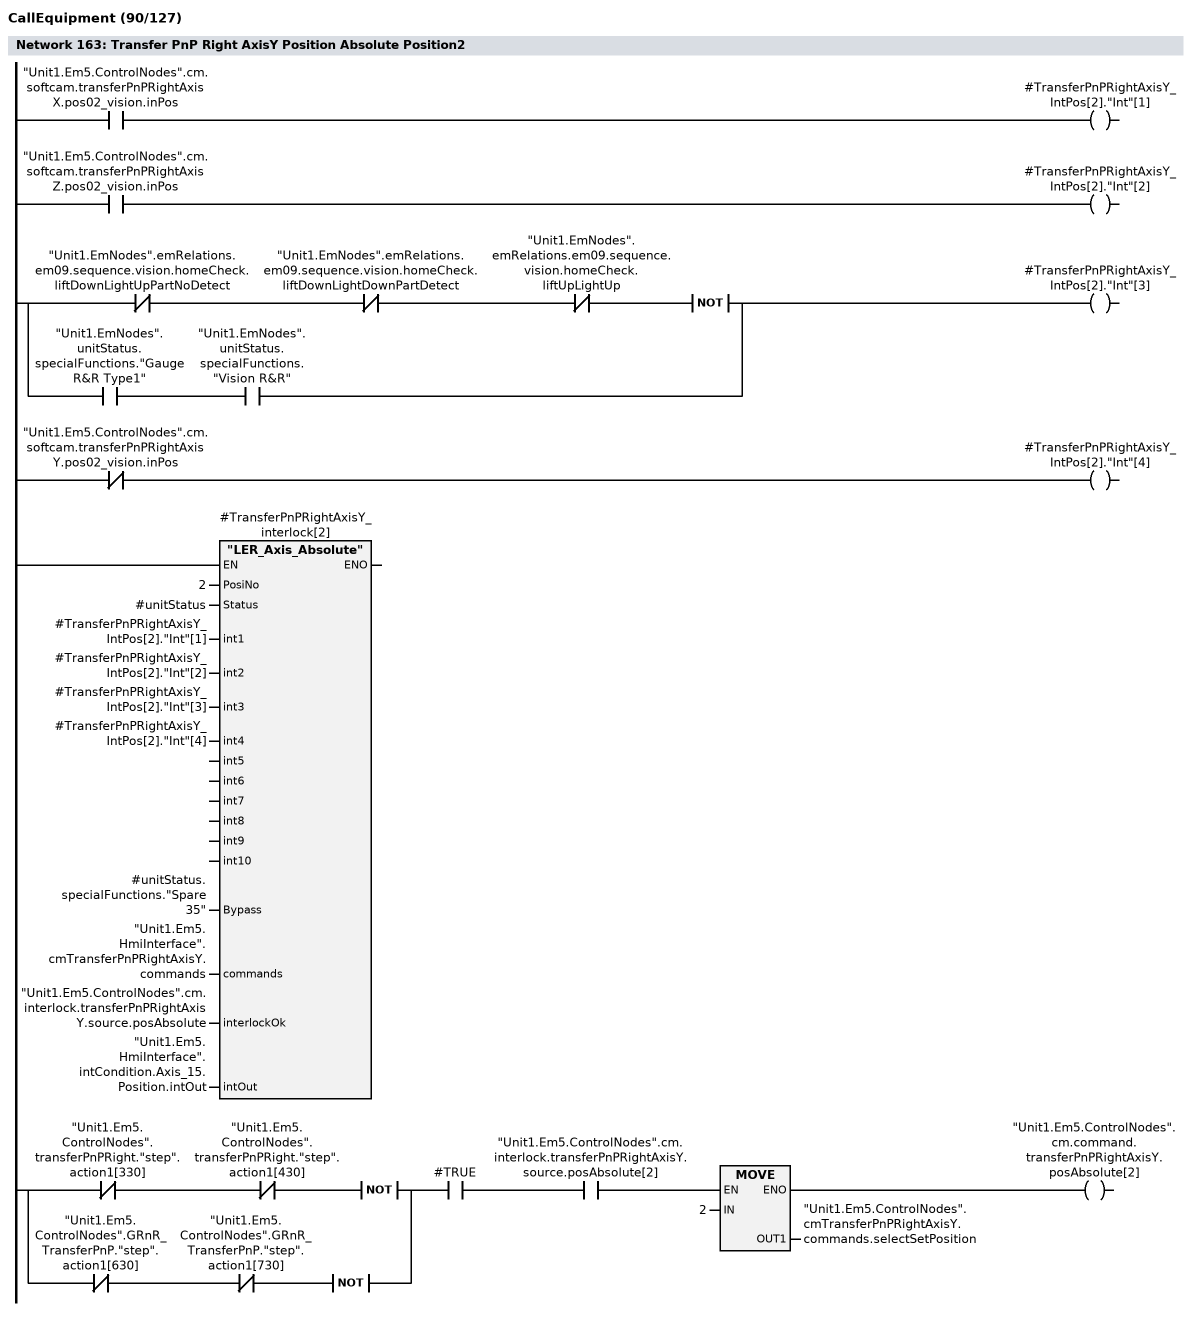
   RUNG wire#powerrail
      Contact( "Unit1.Em5.ControlNodes".cm.softcam.transferPnPRightAxisX.pos02_vision.inPos )
      Coil( #TransferPnPRightAxisY_IntPos[2]."Int"[1] )
   END_RUNG
   RUNG wire#powerrail
      Contact( "Unit1.Em5.ControlNodes".cm.softcam.transferPnPRightAxisZ.pos02_vision.inPos )
      Coil( #TransferPnPRightAxisY_IntPos[2]."Int"[2] )
   END_RUNG
   RUNG wire#powerrail
      I_Contact( "Unit1.EmNodes".emRelations.em09.sequence.vision.homeCheck.liftDownLightUpPartNoDetect )
      I_Contact( "Unit1.EmNodes".emRelations.em09.sequence.vision.homeCheck.liftDownLightDownPartDetect )
      I_Contact( "Unit1.EmNodes".emRelations.em09.sequence.vision.homeCheck.liftUpLightUp )
      Not()
      wire#w1
      Coil( #TransferPnPRightAxisY_IntPos[2]."Int"[3] )
   END_RUNG
   RUNG wire#powerrail
      Contact( "Unit1.EmNodes".unitStatus.specialFunctions."Gauge R&R Type1" )
      Contact( "Unit1.EmNodes".unitStatus.specialFunctions."Vision R&R" )
   END_RUNG wire#w1
   RUNG wire#powerrail
      I_Contact( "Unit1.Em5.ControlNodes".cm.softcam.transferPnPRightAxisY.pos02_vision.inPos )
      Coil( #TransferPnPRightAxisY_IntPos[2]."Int"[4] )
   END_RUNG
   RUNG wire#powerrail
      #TransferPnPRightAxisY_interlock[2](PosiNo := 2, Status := #unitStatus, int1 := #TransferPnPRightAxisY_IntPos[2]."Int"[1], int2 := #TransferPnPRightAxisY_IntPos[2]."Int"[2], int3 := #TransferPnPRightAxisY_IntPos[2]."Int"[3], int4 := #TransferPnPRightAxisY_IntPos[2]."Int"[4], int5 :=, int6 :=, int7 :=, int8 :=, int9 :=, int10 :=, Bypass := #unitStatus.specialFunctions."Spare 35", commands := "Unit1.Em5.HmiInterface".cmTransferPnPRightAxisY.commands, interlockOk := "Unit1.Em5.ControlNodes".cm.interlock.transferPnPRightAxisY.source.posAbsolute, intOut := "Unit1.Em5.HmiInterface".intCondition.Axis_15.Position.intOut)
   END_RUNG
   RUNG wire#powerrail
      I_Contact( "Unit1.Em5.ControlNodes".transferPnPRight."step".action1[330] )
      I_Contact( "Unit1.Em5.ControlNodes".transferPnPRight."step".action1[430] )
      Not()
      wire#w2
      Contact( #TRUE )
      Contact( "Unit1.Em5.ControlNodes".cm.interlock.transferPnPRightAxisY.source.posAbsolute[2] )
      Move(in := 2, out1 => "Unit1.Em5.ControlNodes".cmTransferPnPRightAxisY.commands.selectSetPosition)
      Coil( "Unit1.Em5.ControlNodes".cm.command.transferPnPRightAxisY.posAbsolute[2] )
   END_RUNG
   RUNG wire#powerrail
      I_Contact( "Unit1.Em5.ControlNodes".GRnR_TransferPnP."step".action1[630] )
      I_Contact( "Unit1.Em5.ControlNodes".GRnR_TransferPnP."step".action1[730] )
      Not()
   END_RUNG wire#w2
   // the same network as SCL:
   #TransferPnPRightAxisY_IntPos[2]."Int"[1] := "Unit1.Em5.ControlNodes".cm.softcam.transferPnPRightAxisX.pos02_vision.inPos;
   #TransferPnPRightAxisY_IntPos[2]."Int"[2] := "Unit1.Em5.ControlNodes".cm.softcam.transferPnPRightAxisZ.pos02_vision.inPos;
   #TransferPnPRightAxisY_IntPos[2]."Int"[3] := NOT (NOT "Unit1.EmNodes".emRelations.em09.sequence.vision.homeCheck.liftDownLightUpPartNoDetect AND NOT "Unit1.EmNodes".emRelations.em09.sequence.vision.homeCheck.liftDownLightDownPartDetect AND NOT "Unit1.EmNodes".emRelations.em09.sequence.vision.homeCheck.liftUpLightUp) OR ("Unit1.EmNodes".unitStatus.specialFunctions."Gauge R&R Type1" AND "Unit1.EmNodes".unitStatus.specialFunctions."Vision R&R");
   #TransferPnPRightAxisY_IntPos[2]."Int"[4] := NOT "Unit1.Em5.ControlNodes".cm.softcam.transferPnPRightAxisY.pos02_vision.inPos;
   #TransferPnPRightAxisY_interlock[2](PosiNo := 2,   // "LER_Axis_Absolute"
                           Status := #unitStatus,
                           int1 := #TransferPnPRightAxisY_IntPos[2]."Int"[1],
                           int2 := #TransferPnPRightAxisY_IntPos[2]."Int"[2],
                           int3 := #TransferPnPRightAxisY_IntPos[2]."Int"[3],
                           int4 := #TransferPnPRightAxisY_IntPos[2]."Int"[4],
                           Bypass := #unitStatus.specialFunctions."Spare 35",
                           commands := "Unit1.Em5.HmiInterface".cmTransferPnPRightAxisY.commands,
                           interlockOk := "Unit1.Em5.ControlNodes".cm.interlock.transferPnPRightAxisY.source.posAbsolute,
                           intOut := "Unit1.Em5.HmiInterface".intCondition.Axis_15.Position.intOut);
   #_w1 := (NOT (NOT "Unit1.Em5.ControlNodes".transferPnPRight."step".action1[330] AND NOT "Unit1.Em5.ControlNodes".transferPnPRight."step".action1[430]) OR NOT (NOT "Unit1.Em5.ControlNodes".GRnR_TransferPnP."step".action1[630] AND NOT "Unit1.Em5.ControlNodes".GRnR_TransferPnP."step".action1[730])) AND #TRUE AND "Unit1.Em5.ControlNodes".cm.interlock.transferPnPRightAxisY.source.posAbsolute[2];
   IF #_w1 THEN "Unit1.Em5.ControlNodes".cmTransferPnPRightAxisY.commands.selectSetPosition := 2; END_IF;
   "Unit1.Em5.ControlNodes".cm.command.transferPnPRightAxisY.posAbsolute[2] := #_w1;
END_REGION

REGION Network 164: Transfer PnP Right AxisY Position Absolute Position3
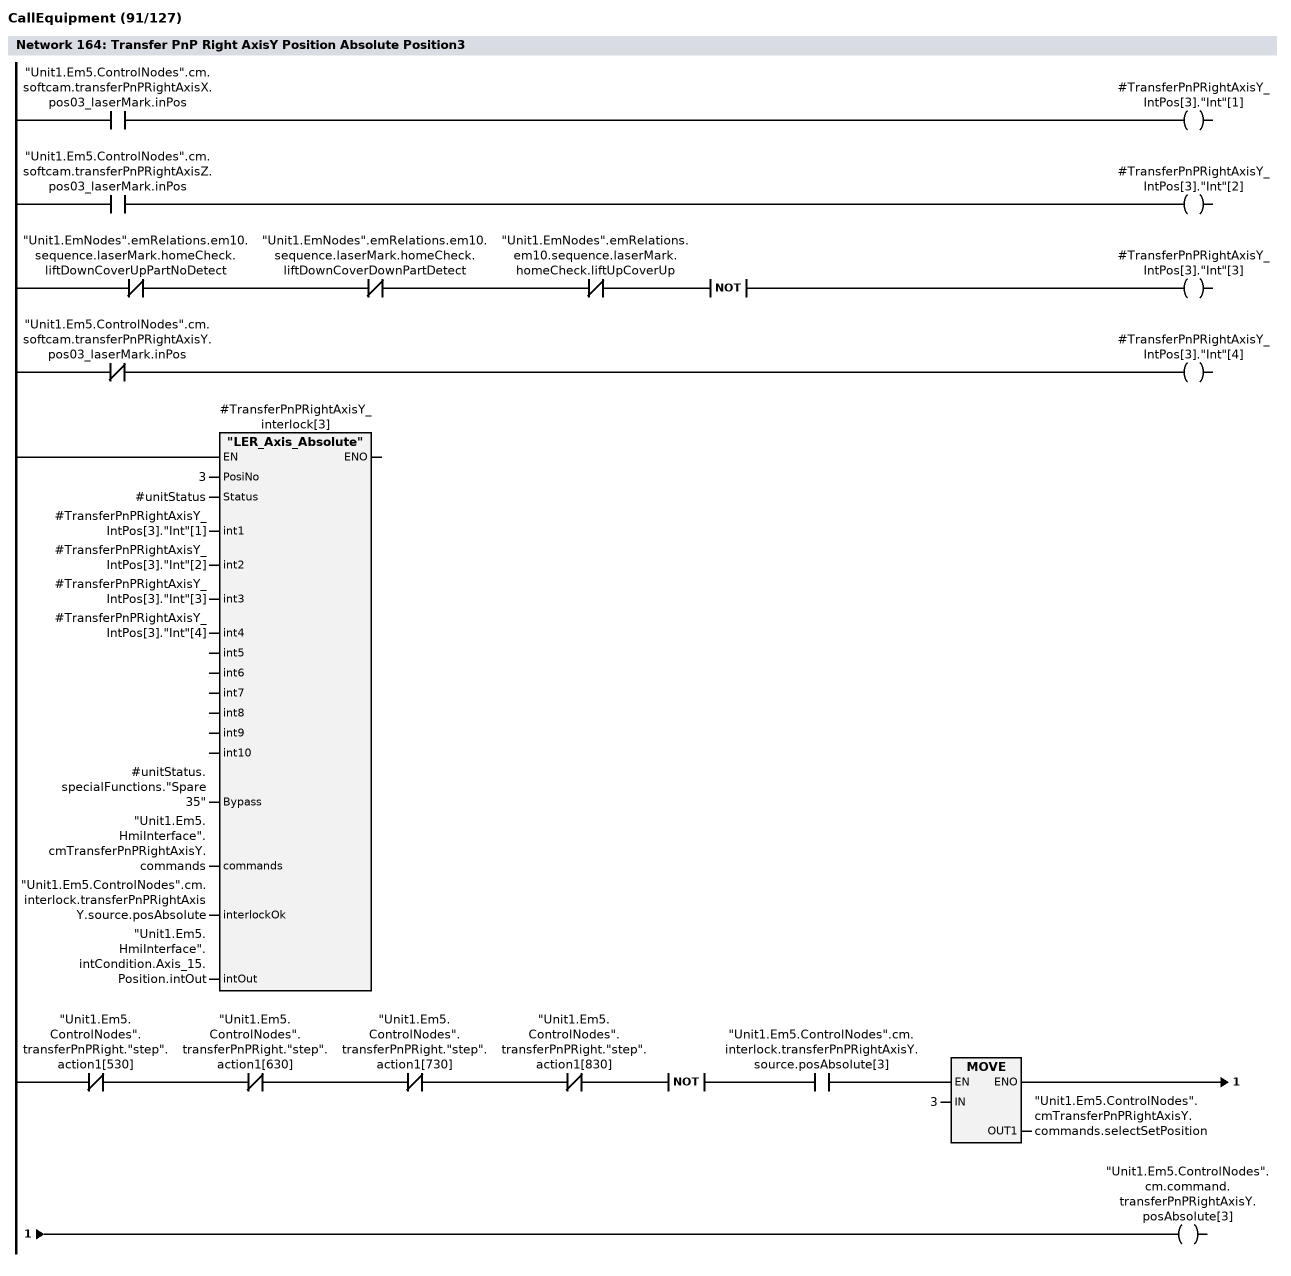
   RUNG wire#powerrail
      Contact( "Unit1.Em5.ControlNodes".cm.softcam.transferPnPRightAxisX.pos03_laserMark.inPos )
      Coil( #TransferPnPRightAxisY_IntPos[3]."Int"[1] )
   END_RUNG
   RUNG wire#powerrail
      Contact( "Unit1.Em5.ControlNodes".cm.softcam.transferPnPRightAxisZ.pos03_laserMark.inPos )
      Coil( #TransferPnPRightAxisY_IntPos[3]."Int"[2] )
   END_RUNG
   RUNG wire#powerrail
      I_Contact( "Unit1.EmNodes".emRelations.em10.sequence.laserMark.homeCheck.liftDownCoverUpPartNoDetect )
      I_Contact( "Unit1.EmNodes".emRelations.em10.sequence.laserMark.homeCheck.liftDownCoverDownPartDetect )
      I_Contact( "Unit1.EmNodes".emRelations.em10.sequence.laserMark.homeCheck.liftUpCoverUp )
      Not()
      Coil( #TransferPnPRightAxisY_IntPos[3]."Int"[3] )
   END_RUNG
   RUNG wire#powerrail
      I_Contact( "Unit1.Em5.ControlNodes".cm.softcam.transferPnPRightAxisY.pos03_laserMark.inPos )
      Coil( #TransferPnPRightAxisY_IntPos[3]."Int"[4] )
   END_RUNG
   RUNG wire#powerrail
      #TransferPnPRightAxisY_interlock[3](PosiNo := 3, Status := #unitStatus, int1 := #TransferPnPRightAxisY_IntPos[3]."Int"[1], int2 := #TransferPnPRightAxisY_IntPos[3]."Int"[2], int3 := #TransferPnPRightAxisY_IntPos[3]."Int"[3], int4 := #TransferPnPRightAxisY_IntPos[3]."Int"[4], int5 :=, int6 :=, int7 :=, int8 :=, int9 :=, int10 :=, Bypass := #unitStatus.specialFunctions."Spare 35", commands := "Unit1.Em5.HmiInterface".cmTransferPnPRightAxisY.commands, interlockOk := "Unit1.Em5.ControlNodes".cm.interlock.transferPnPRightAxisY.source.posAbsolute, intOut := "Unit1.Em5.HmiInterface".intCondition.Axis_15.Position.intOut)
   END_RUNG
   RUNG wire#powerrail
      I_Contact( "Unit1.Em5.ControlNodes".transferPnPRight."step".action1[530] )
      I_Contact( "Unit1.Em5.ControlNodes".transferPnPRight."step".action1[630] )
      I_Contact( "Unit1.Em5.ControlNodes".transferPnPRight."step".action1[730] )
      I_Contact( "Unit1.Em5.ControlNodes".transferPnPRight."step".action1[830] )
      Not()
      Contact( "Unit1.Em5.ControlNodes".cm.interlock.transferPnPRightAxisY.source.posAbsolute[3] )
      Move(in := 3, out1 => "Unit1.Em5.ControlNodes".cmTransferPnPRightAxisY.commands.selectSetPosition)
      Coil( "Unit1.Em5.ControlNodes".cm.command.transferPnPRightAxisY.posAbsolute[3] )
   END_RUNG
   // the same network as SCL:
   #TransferPnPRightAxisY_IntPos[3]."Int"[1] := "Unit1.Em5.ControlNodes".cm.softcam.transferPnPRightAxisX.pos03_laserMark.inPos;
   #TransferPnPRightAxisY_IntPos[3]."Int"[2] := "Unit1.Em5.ControlNodes".cm.softcam.transferPnPRightAxisZ.pos03_laserMark.inPos;
   #TransferPnPRightAxisY_IntPos[3]."Int"[3] := NOT (NOT "Unit1.EmNodes".emRelations.em10.sequence.laserMark.homeCheck.liftDownCoverUpPartNoDetect AND NOT "Unit1.EmNodes".emRelations.em10.sequence.laserMark.homeCheck.liftDownCoverDownPartDetect AND NOT "Unit1.EmNodes".emRelations.em10.sequence.laserMark.homeCheck.liftUpCoverUp);
   #TransferPnPRightAxisY_IntPos[3]."Int"[4] := NOT "Unit1.Em5.ControlNodes".cm.softcam.transferPnPRightAxisY.pos03_laserMark.inPos;
   #TransferPnPRightAxisY_interlock[3](PosiNo := 3,   // "LER_Axis_Absolute"
                           Status := #unitStatus,
                           int1 := #TransferPnPRightAxisY_IntPos[3]."Int"[1],
                           int2 := #TransferPnPRightAxisY_IntPos[3]."Int"[2],
                           int3 := #TransferPnPRightAxisY_IntPos[3]."Int"[3],
                           int4 := #TransferPnPRightAxisY_IntPos[3]."Int"[4],
                           Bypass := #unitStatus.specialFunctions."Spare 35",
                           commands := "Unit1.Em5.HmiInterface".cmTransferPnPRightAxisY.commands,
                           interlockOk := "Unit1.Em5.ControlNodes".cm.interlock.transferPnPRightAxisY.source.posAbsolute,
                           intOut := "Unit1.Em5.HmiInterface".intCondition.Axis_15.Position.intOut);
   #_w1 := NOT (NOT "Unit1.Em5.ControlNodes".transferPnPRight."step".action1[530] AND NOT "Unit1.Em5.ControlNodes".transferPnPRight."step".action1[630] AND NOT "Unit1.Em5.ControlNodes".transferPnPRight."step".action1[730] AND NOT "Unit1.Em5.ControlNodes".transferPnPRight."step".action1[830]) AND "Unit1.Em5.ControlNodes".cm.interlock.transferPnPRightAxisY.source.posAbsolute[3];
   IF #_w1 THEN "Unit1.Em5.ControlNodes".cmTransferPnPRightAxisY.commands.selectSetPosition := 3; END_IF;
   "Unit1.Em5.ControlNodes".cm.command.transferPnPRightAxisY.posAbsolute[3] := #_w1;
END_REGION

REGION Network 165: Transfer PnP Right AxisY Position Absolute Position4
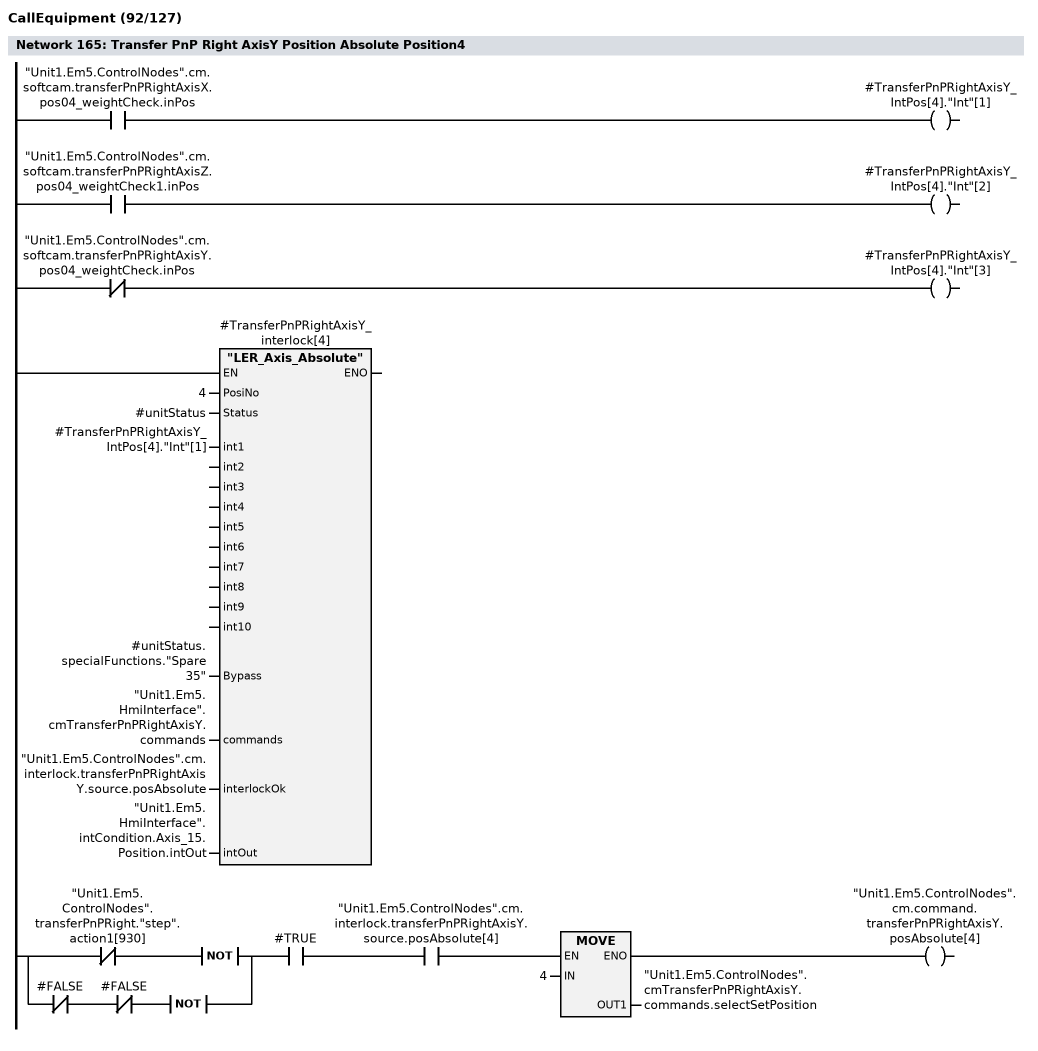
   RUNG wire#powerrail
      Contact( "Unit1.Em5.ControlNodes".cm.softcam.transferPnPRightAxisX.pos04_weightCheck.inPos )
      Coil( #TransferPnPRightAxisY_IntPos[4]."Int"[1] )
   END_RUNG
   RUNG wire#powerrail
      Contact( "Unit1.Em5.ControlNodes".cm.softcam.transferPnPRightAxisZ.pos04_weightCheck1.inPos )
      Coil( #TransferPnPRightAxisY_IntPos[4]."Int"[2] )
   END_RUNG
   RUNG wire#powerrail
      I_Contact( "Unit1.Em5.ControlNodes".cm.softcam.transferPnPRightAxisY.pos04_weightCheck.inPos )
      Coil( #TransferPnPRightAxisY_IntPos[4]."Int"[3] )
   END_RUNG
   RUNG wire#powerrail
      #TransferPnPRightAxisY_interlock[4](PosiNo := 4, Status := #unitStatus, int1 := #TransferPnPRightAxisY_IntPos[4]."Int"[1], int2 :=, int3 :=, int4 :=, int5 :=, int6 :=, int7 :=, int8 :=, int9 :=, int10 :=, Bypass := #unitStatus.specialFunctions."Spare 35", commands := "Unit1.Em5.HmiInterface".cmTransferPnPRightAxisY.commands, interlockOk := "Unit1.Em5.ControlNodes".cm.interlock.transferPnPRightAxisY.source.posAbsolute, intOut := "Unit1.Em5.HmiInterface".intCondition.Axis_15.Position.intOut)
   END_RUNG
   RUNG wire#powerrail
      I_Contact( "Unit1.Em5.ControlNodes".transferPnPRight."step".action1[930] )
      Not()
      wire#w1
      Contact( #TRUE )
      Contact( "Unit1.Em5.ControlNodes".cm.interlock.transferPnPRightAxisY.source.posAbsolute[4] )
      Move(in := 4, out1 => "Unit1.Em5.ControlNodes".cmTransferPnPRightAxisY.commands.selectSetPosition)
      Coil( "Unit1.Em5.ControlNodes".cm.command.transferPnPRightAxisY.posAbsolute[4] )
   END_RUNG
   RUNG wire#powerrail
      I_Contact( #FALSE )
      I_Contact( #FALSE )
      Not()
   END_RUNG wire#w1
   // the same network as SCL:
   #TransferPnPRightAxisY_IntPos[4]."Int"[1] := "Unit1.Em5.ControlNodes".cm.softcam.transferPnPRightAxisX.pos04_weightCheck.inPos;
   #TransferPnPRightAxisY_IntPos[4]."Int"[2] := "Unit1.Em5.ControlNodes".cm.softcam.transferPnPRightAxisZ.pos04_weightCheck1.inPos;
   #TransferPnPRightAxisY_IntPos[4]."Int"[3] := NOT "Unit1.Em5.ControlNodes".cm.softcam.transferPnPRightAxisY.pos04_weightCheck.inPos;
   #TransferPnPRightAxisY_interlock[4](PosiNo := 4,   // "LER_Axis_Absolute"
                           Status := #unitStatus,
                           int1 := #TransferPnPRightAxisY_IntPos[4]."Int"[1],
                           Bypass := #unitStatus.specialFunctions."Spare 35",
                           commands := "Unit1.Em5.HmiInterface".cmTransferPnPRightAxisY.commands,
                           interlockOk := "Unit1.Em5.ControlNodes".cm.interlock.transferPnPRightAxisY.source.posAbsolute,
                           intOut := "Unit1.Em5.HmiInterface".intCondition.Axis_15.Position.intOut);
   #_w1 := (NOT (NOT "Unit1.Em5.ControlNodes".transferPnPRight."step".action1[930]) OR NOT (NOT #FALSE AND NOT #FALSE)) AND #TRUE AND "Unit1.Em5.ControlNodes".cm.interlock.transferPnPRightAxisY.source.posAbsolute[4];
   IF #_w1 THEN "Unit1.Em5.ControlNodes".cmTransferPnPRightAxisY.commands.selectSetPosition := 4; END_IF;
   "Unit1.Em5.ControlNodes".cm.command.transferPnPRightAxisY.posAbsolute[4] := #_w1;
END_REGION

REGION Network 166: Transfer PnP Right AxisY Position Absolute Position5
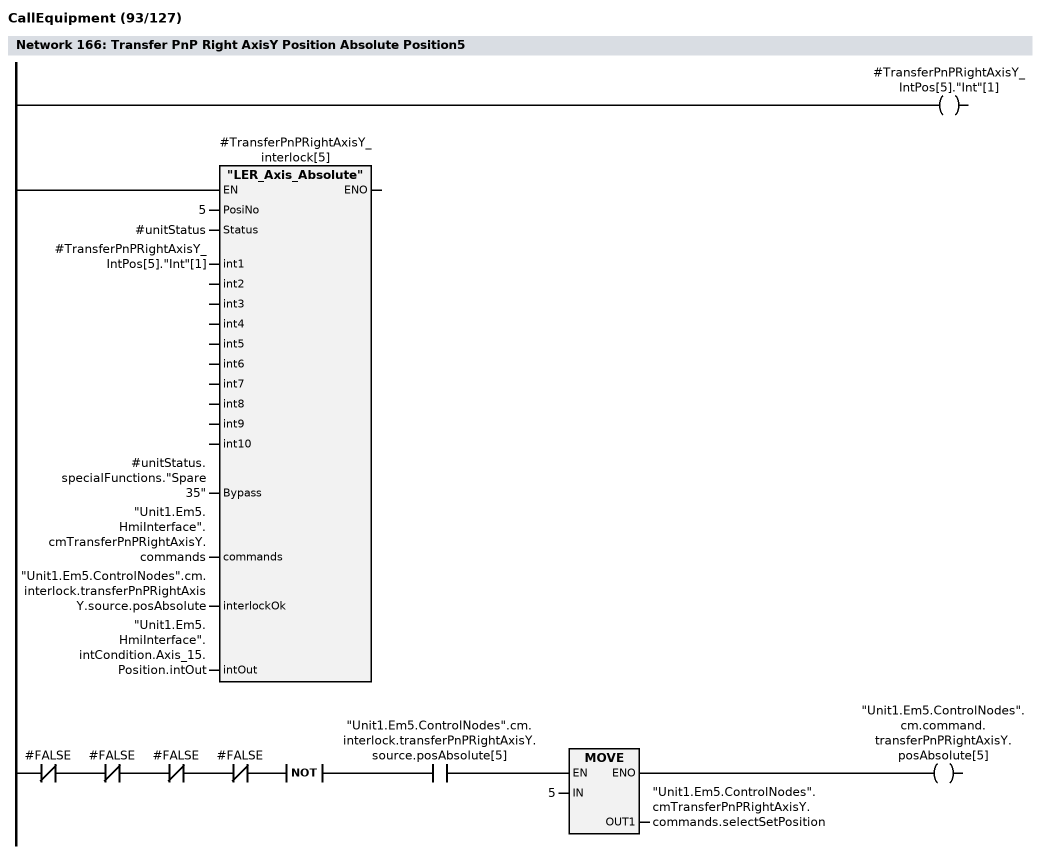
   RUNG wire#powerrail
      Coil( #TransferPnPRightAxisY_IntPos[5]."Int"[1] )
   END_RUNG
   RUNG wire#powerrail
      #TransferPnPRightAxisY_interlock[5](PosiNo := 5, Status := #unitStatus, int1 := #TransferPnPRightAxisY_IntPos[5]."Int"[1], int2 :=, int3 :=, int4 :=, int5 :=, int6 :=, int7 :=, int8 :=, int9 :=, int10 :=, Bypass := #unitStatus.specialFunctions."Spare 35", commands := "Unit1.Em5.HmiInterface".cmTransferPnPRightAxisY.commands, interlockOk := "Unit1.Em5.ControlNodes".cm.interlock.transferPnPRightAxisY.source.posAbsolute, intOut := "Unit1.Em5.HmiInterface".intCondition.Axis_15.Position.intOut)
   END_RUNG
   RUNG wire#powerrail
      I_Contact( #FALSE )
      I_Contact( #FALSE )
      I_Contact( #FALSE )
      I_Contact( #FALSE )
      Not()
      Contact( "Unit1.Em5.ControlNodes".cm.interlock.transferPnPRightAxisY.source.posAbsolute[5] )
      Move(in := 5, out1 => "Unit1.Em5.ControlNodes".cmTransferPnPRightAxisY.commands.selectSetPosition)
      Coil( "Unit1.Em5.ControlNodes".cm.command.transferPnPRightAxisY.posAbsolute[5] )
   END_RUNG
   // the same network as SCL:
   #TransferPnPRightAxisY_IntPos[5]."Int"[1] := TRUE;
   #TransferPnPRightAxisY_interlock[5](PosiNo := 5,   // "LER_Axis_Absolute"
                           Status := #unitStatus,
                           int1 := #TransferPnPRightAxisY_IntPos[5]."Int"[1],
                           Bypass := #unitStatus.specialFunctions."Spare 35",
                           commands := "Unit1.Em5.HmiInterface".cmTransferPnPRightAxisY.commands,
                           interlockOk := "Unit1.Em5.ControlNodes".cm.interlock.transferPnPRightAxisY.source.posAbsolute,
                           intOut := "Unit1.Em5.HmiInterface".intCondition.Axis_15.Position.intOut);
   #_w1 := NOT (NOT #FALSE AND NOT #FALSE AND NOT #FALSE AND NOT #FALSE) AND "Unit1.Em5.ControlNodes".cm.interlock.transferPnPRightAxisY.source.posAbsolute[5];
   IF #_w1 THEN "Unit1.Em5.ControlNodes".cmTransferPnPRightAxisY.commands.selectSetPosition := 5; END_IF;
   "Unit1.Em5.ControlNodes".cm.command.transferPnPRightAxisY.posAbsolute[5] := #_w1;
END_REGION

REGION Network 167: Transfer PnP Right AxisY Position Absolute Position7
